   1:  PR[GP1:91,2] = PR[GP1:90,2] + -18.004;
   1:L PR[91] R[100]mm/sec CNT100;
   1:  PR[GP1:91,1] = PR[GP1:90,1] + -44.967;
   1:  PR[GP1:91,2] = PR[GP1:90,2] + -27.584;
   1:L PR[91] R[100]mm/sec CNT100;
   1:  PR[GP1:91,1] = PR[GP1:90,1] + -42.334;
   1:  PR[GP1:91,2] = PR[GP1:90,2] + -29.755;
   1:L PR[91] R[100]mm/sec CNT100;
   1:  PR[GP1:91,1] = PR[GP1:90,1] + -32.989;
   1:  PR[GP1:91,2] = PR[GP1:90,2] + -37.151;
   1:L PR[91] R[100]mm/sec CNT100;
   1:  PR[GP1:91,1] = PR[GP1:90,1] + -30.364;
   1:  PR[GP1:91,2] = PR[GP1:90,2] + -38.119;
   1:L PR[91] R[100]mm/sec CNT100;
   1:  PR[GP1:91,1] = PR[GP1:90,1] + -18.205;
   1:  PR[GP1:91,2] = PR[GP1:90,2] + -42.108;
   1:L PR[91] R[100]mm/sec CNT100;
   1:  PR[GP1:91,1] = PR[GP1:90,1] + -16.121;
   1:  PR[GP1:91,2] = PR[GP1:90,2] + -42.145;
   1:L PR[91] R[100]mm/sec CNT100;
   1:  PR[GP1:91,1] = PR[GP1:90,1] + -2.431;
   1:  PR[GP1:91,2] = PR[GP1:90,2] + -41.656;
   1:L PR[91] R[100]mm/sec CNT100;
   1:  PR[GP1:91,1] = PR[GP1:90,1] + -1.102;
   1:  PR[GP1:91,2] = PR[GP1:90,2] + -41.254;
   1:L PR[91] R[100]mm/sec CNT100;
   1:  PR[GP1:91,1] = PR[GP1:90,1] + 1.318;
   1:L PR[91] R[100]mm/sec CNT100;
   1:  PR[GP1:91,1] = PR[GP1:90,1] + 2.646;
   1:  PR[GP1:91,2] = PR[GP1:90,2] + -41.656;
   1:L PR[91] R[100]mm/sec CNT100;
   1:  PR[GP1:91,1] = PR[GP1:90,1] + 16.336;
   1:  PR[GP1:91,2] = PR[GP1:90,2] + -42.144;
   1:L PR[91] R[100]mm/sec CNT100;
   1:  PR[GP1:91,1] = PR[GP1:90,1] + 18.420;
   1:  PR[GP1:91,2] = PR[GP1:90,2] + -42.107;
   1:L PR[91] R[100]mm/sec CNT100;
   1:  PR[GP1:91,1] = PR[GP1:90,1] + 30.578;
   1:  PR[GP1:91,2] = PR[GP1:90,2] + -38.119;
   1:L PR[91] R[100]mm/sec CNT100;
   1:  PR[GP1:91,1] = PR[GP1:90,1] + 33.204;
   1:  PR[GP1:91,2] = PR[GP1:90,2] + -37.151;
   1:L PR[91] R[100]mm/sec CNT100;
   1:  PR[GP1:91,1] = PR[GP1:90,1] + 42.548;
   1:  PR[GP1:91,2] = PR[GP1:90,2] + -29.754;
   1:L PR[91] R[100]mm/sec CNT100;
   1:  PR[GP1:91,1] = PR[GP1:90,1] + 45.181;
   1:  PR[GP1:91,2] = PR[GP1:90,2] + -27.580;
   1:L PR[91] R[100]mm/sec CNT100;
   1:  PR[GP1:91,1] = PR[GP1:90,1] + 50.972;
   1:  PR[GP1:91,2] = PR[GP1:90,2] + -18.005;
   1:L PR[91] R[100]mm/sec CNT100;
   1:  PR[GP1:91,1] = PR[GP1:90,1] + 52.939;
   1:  PR[GP1:91,2] = PR[GP1:90,2] + -14.686;
   1:L PR[91] R[100]mm/sec CNT100;
   1:  PR[GP1:91,1] = PR[GP1:90,1] + 53.674;
   1:  PR[GP1:91,2] = PR[GP1:90,2] + -10.625;
   1:L PR[91] R[100]mm/sec CNT100;
   1:  PR[GP1:91,1] = PR[GP1:90,1] + 54.569;
   1:  PR[GP1:91,2] = PR[GP1:90,2] + -5.071;
   1:L PR[91] R[100]mm/sec CNT100;
   1:  PR[GP1:91,1] = PR[GP1:90,1] + 55.491;
   1:  PR[GP1:91,2] = PR[GP1:90,2] + -0.062;
   1:L PR[91] R[100]mm/sec CNT100;
   1:  PR[GP1:91,1] = PR[GP1:90,1] + 54.883;
   1:  PR[GP1:91,2] = PR[GP1:90,2] + 4.006;
   1:L PR[91] R[100]mm/sec CNT100;
   1:  PR[GP1:91,1] = PR[GP1:90,1] + 52.939;
   1:  PR[GP1:91,2] = PR[GP1:90,2] + 14.540;
   1:L PR[91] R[100]mm/sec CNT100;
   1:  PR[GP1:91,1] = PR[GP1:90,1] + 50.974;
   1:  PR[GP1:91,2] = PR[GP1:90,2] + 17.860;
   1:L PR[91] R[100]mm/sec CNT100;
   1:  PR[GP1:91,1] = PR[GP1:90,1] + 45.181;
   1:  PR[GP1:91,2] = PR[GP1:90,2] + 27.435;
   1:L PR[91] R[100]mm/sec CNT100;
   1:  PR[GP1:91,1] = PR[GP1:90,1] + 42.550;
   1:  PR[GP1:91,2] = PR[GP1:90,2] + 29.610;
   1:L PR[91] R[100]mm/sec CNT100;
   1:  PR[GP1:91,1] = PR[GP1:90,1] + 33.204;
   1:  PR[GP1:91,2] = PR[GP1:90,2] + 37.007;
   1:L PR[91] R[100]mm/sec CNT100;
   1:  PR[GP1:91,1] = PR[GP1:90,1] + 30.579;
   1:  PR[GP1:91,2] = PR[GP1:90,2] + 37.975;
   1:L PR[91] R[100]mm/sec CNT100;
   1:  PR[GP1:91,1] = PR[GP1:90,1] + 18.419;
   1:  PR[GP1:91,2] = PR[GP1:90,2] + 41.964;
   1:L PR[91] R[100]mm/sec CNT100;
   1:  PR[GP1:91,1] = PR[GP1:90,1] + 16.336;
   1:  PR[GP1:91,2] = PR[GP1:90,2] + 42.001;
   1:L PR[91] R[100]mm/sec CNT100;
   1:  PR[GP1:91,1] = PR[GP1:90,1] + 2.640;
   1:  PR[GP1:91,2] = PR[GP1:90,2] + 41.510;
   1:L PR[91] R[100]mm/sec CNT100;
   1:  PR[GP1:91,1] = PR[GP1:90,1] + 1.317;
   1:  PR[GP1:91,2] = PR[GP1:90,2] + 41.113;
   1:L PR[91] R[100]mm/sec CNT100;
   1:  ! -- Layer/Ebene 159 -- !;
   1:  PR[91] = PR[90];
   1:  PR[GP1:91,1] = PR[GP1:90,1] + -1.075;
   1:  PR[GP1:91,2] = PR[GP1:90,2] + 41.286;
   1:  PR[GP1:91,3] = PR[GP1:90,3] + 97.295;
   1:L PR[91] R[100]mm/sec CNT100;
   1:  PR[GP1:91,1] = PR[GP1:90,1] + -2.125;
   1:  PR[GP1:91,2] = PR[GP1:90,2] + 41.599;
   1:L PR[91] R[100]mm/sec CNT100;
   1:  PR[GP1:91,1] = PR[GP1:90,1] + -16.159;
   1:  PR[GP1:91,2] = PR[GP1:90,2] + 42.102;
   1:L PR[91] R[100]mm/sec CNT100;
   1:  PR[GP1:91,1] = PR[GP1:90,1] + -17.943;
   1:  PR[GP1:91,2] = PR[GP1:90,2] + 42.070;
   1:L PR[91] R[100]mm/sec CNT100;
   1:  PR[GP1:91,1] = PR[GP1:90,1] + -30.434;
   1:  PR[GP1:91,2] = PR[GP1:90,2] + 37.973;
   1:L PR[91] R[100]mm/sec CNT100;
   1:  PR[GP1:91,1] = PR[GP1:90,1] + -32.768;
   1:  PR[GP1:91,2] = PR[GP1:90,2] + 37.112;
   1:L PR[91] R[100]mm/sec CNT100;
   1:  PR[GP1:91,1] = PR[GP1:90,1] + -42.396;
   1:  PR[GP1:91,2] = PR[GP1:90,2] + 29.493;
   1:L PR[91] R[100]mm/sec CNT100;
   1:  PR[GP1:91,1] = PR[GP1:90,1] + -44.783;
   1:  PR[GP1:91,2] = PR[GP1:90,2] + 27.523;
   1:L PR[91] R[100]mm/sec CNT100;
   1:  PR[GP1:91,1] = PR[GP1:90,1] + -50.767;
   1:  PR[GP1:91,2] = PR[GP1:90,2] + 17.626;
   1:L PR[91] R[100]mm/sec CNT100;
   1:  PR[GP1:91,1] = PR[GP1:90,1] + -52.567;
   1:  PR[GP1:91,2] = PR[GP1:90,2] + 14.580;
   1:L PR[91] R[100]mm/sec CNT100;
   1:  PR[GP1:91,1] = PR[GP1:90,1] + -53.240;
   1:  PR[GP1:91,2] = PR[GP1:90,2] + 10.867;
   1:L PR[91] R[100]mm/sec CNT100;
   1:  PR[GP1:91,1] = PR[GP1:90,1] + -54.062;
   1:  PR[GP1:91,2] = PR[GP1:90,2] + 5.768;
   1:L PR[91] R[100]mm/sec CNT100;
   1:  PR[GP1:91,1] = PR[GP1:90,1] + -55.139;
   1:  PR[GP1:91,2] = PR[GP1:90,2] + -0.082;
   1:L PR[91] R[100]mm/sec CNT100;
   1:  PR[GP1:91,1] = PR[GP1:90,1] + -54.579;
   1:  PR[GP1:91,2] = PR[GP1:90,2] + -3.819;
   1:L PR[91] R[100]mm/sec CNT100;
   1:  PR[GP1:91,1] = PR[GP1:90,1] + -52.567;
   1:  PR[GP1:91,2] = PR[GP1:90,2] + -14.723;
   1:L PR[91] R[100]mm/sec CNT100;
   1:  PR[GP1:91,1] = PR[GP1:90,1] + -50.766;
   1:  PR[GP1:91,2] = PR[GP1:90,2] + -17.771;
   1:L PR[91] R[100]mm/sec CNT100;
   1:  PR[GP1:91,1] = PR[GP1:90,1] + -44.782;
   1:  PR[GP1:91,2] = PR[GP1:90,2] + -27.668;
   1:L PR[91] R[100]mm/sec CNT100;
   1:  PR[GP1:91,1] = PR[GP1:90,1] + -42.395;
   1:  PR[GP1:91,2] = PR[GP1:90,2] + -29.637;
   1:L PR[91] R[100]mm/sec CNT100;
   1:  PR[GP1:91,1] = PR[GP1:90,1] + -32.768;
   1:  PR[GP1:91,2] = PR[GP1:90,2] + -37.256;
   1:L PR[91] R[100]mm/sec CNT100;
   1:  PR[GP1:91,1] = PR[GP1:90,1] + -30.433;
   1:  PR[GP1:91,2] = PR[GP1:90,2] + -38.117;
   1:L PR[91] R[100]mm/sec CNT100;
   1:  PR[GP1:91,1] = PR[GP1:90,1] + -17.944;
   1:  PR[GP1:91,2] = PR[GP1:90,2] + -42.214;
   1:L PR[91] R[100]mm/sec CNT100;
   1:  PR[GP1:91,1] = PR[GP1:90,1] + -16.160;
   1:  PR[GP1:91,2] = PR[GP1:90,2] + -42.245;
   1:L PR[91] R[100]mm/sec CNT100;
   1:  PR[GP1:91,1] = PR[GP1:90,1] + -2.133;
   1:  PR[GP1:91,2] = PR[GP1:90,2] + -41.745;
   1:L PR[91] R[100]mm/sec CNT100;
   1:  PR[GP1:91,1] = PR[GP1:90,1] + -1.076;
   1:  PR[GP1:91,2] = PR[GP1:90,2] + -41.428;
   1:L PR[91] R[100]mm/sec CNT100;
   1:  PR[GP1:91,1] = PR[GP1:90,1] + 1.292;
   1:L PR[91] R[100]mm/sec CNT100;
   1:  PR[GP1:91,1] = PR[GP1:90,1] + 2.349;
   1:  PR[GP1:91,2] = PR[GP1:90,2] + -41.745;
   1:L PR[91] R[100]mm/sec CNT100;
   1:  PR[GP1:91,1] = PR[GP1:90,1] + 16.375;
   1:  PR[GP1:91,2] = PR[GP1:90,2] + -42.245;
   1:L PR[91] R[100]mm/sec CNT100;
   1:  PR[GP1:91,1] = PR[GP1:90,1] + 18.159;
   1:  PR[GP1:91,2] = PR[GP1:90,2] + -42.214;
   1:L PR[91] R[100]mm/sec CNT100;
   1:  PR[GP1:91,1] = PR[GP1:90,1] + 30.647;
   1:  PR[GP1:91,2] = PR[GP1:90,2] + -38.116;
   1:L PR[91] R[100]mm/sec CNT100;
   1:  PR[GP1:91,1] = PR[GP1:90,1] + 32.982;
   1:  PR[GP1:91,2] = PR[GP1:90,2] + -37.256;
   1:L PR[91] R[100]mm/sec CNT100;
   1:  PR[GP1:91,1] = PR[GP1:90,1] + 42.608;
   1:  PR[GP1:91,2] = PR[GP1:90,2] + -29.636;
   1:L PR[91] R[100]mm/sec CNT100;
   1:  PR[GP1:91,1] = PR[GP1:90,1] + 44.996;
   1:  PR[GP1:91,2] = PR[GP1:90,2] + -27.664;
   1:L PR[91] R[100]mm/sec CNT100;
   1:  PR[GP1:91,1] = PR[GP1:90,1] + 50.980;
   1:  PR[GP1:91,2] = PR[GP1:90,2] + -17.772;
   1:L PR[91] R[100]mm/sec CNT100;
   1:  PR[GP1:91,1] = PR[GP1:90,1] + 52.780;
   1:  PR[GP1:91,2] = PR[GP1:90,2] + -14.733;
   1:L PR[91] R[100]mm/sec CNT100;
   1:  PR[GP1:91,1] = PR[GP1:90,1] + 53.454;
   1:  PR[GP1:91,2] = PR[GP1:90,2] + -11.014;
   1:L PR[91] R[100]mm/sec CNT100;
   1:  PR[GP1:91,1] = PR[GP1:90,1] + 54.276;
   1:  PR[GP1:91,2] = PR[GP1:90,2] + -5.913;
   1:L PR[91] R[100]mm/sec CNT100;
   1:  PR[GP1:91,1] = PR[GP1:90,1] + 55.352;
   1:  PR[GP1:91,2] = PR[GP1:90,2] + -0.062;
   1:L PR[91] R[100]mm/sec CNT100;
   1:  PR[GP1:91,1] = PR[GP1:90,1] + 54.793;
   1:  PR[GP1:91,2] = PR[GP1:90,2] + 3.680;
   1:L PR[91] R[100]mm/sec CNT100;
   1:  PR[GP1:91,1] = PR[GP1:90,1] + 52.781;
   1:  PR[GP1:91,2] = PR[GP1:90,2] + 14.587;
   1:L PR[91] R[100]mm/sec CNT100;
   1:  PR[GP1:91,1] = PR[GP1:90,1] + 50.981;
   1:  PR[GP1:91,2] = PR[GP1:90,2] + 17.627;
   1:L PR[91] R[100]mm/sec CNT100;
   1:  PR[GP1:91,1] = PR[GP1:90,1] + 44.997;
   1:  PR[GP1:91,2] = PR[GP1:90,2] + 27.520;
   1:L PR[91] R[100]mm/sec CNT100;
   1:  PR[GP1:91,1] = PR[GP1:90,1] + 42.609;
   1:  PR[GP1:91,2] = PR[GP1:90,2] + 29.492;
   1:L PR[91] R[100]mm/sec CNT100;
   1:  PR[GP1:91,1] = PR[GP1:90,1] + 32.982;
   1:  PR[GP1:91,2] = PR[GP1:90,2] + 37.112;
   1:L PR[91] R[100]mm/sec CNT100;
   1:  PR[GP1:91,1] = PR[GP1:90,1] + 30.648;
   1:  PR[GP1:91,2] = PR[GP1:90,2] + 37.973;
   1:L PR[91] R[100]mm/sec CNT100;
   1:  PR[GP1:91,1] = PR[GP1:90,1] + 18.158;
   1:  PR[GP1:91,2] = PR[GP1:90,2] + 42.070;
   1:L PR[91] R[100]mm/sec CNT100;
   1:  PR[GP1:91,1] = PR[GP1:90,1] + 16.374;
   1:  PR[GP1:91,2] = PR[GP1:90,2] + 42.102;
   1:L PR[91] R[100]mm/sec CNT100;
   1:  PR[GP1:91,1] = PR[GP1:90,1] + 2.341;
   1:  PR[GP1:91,2] = PR[GP1:90,2] + 41.599;
   1:L PR[91] R[100]mm/sec CNT100;
   1:  PR[GP1:91,1] = PR[GP1:90,1] + 1.291;
   1:  PR[GP1:91,2] = PR[GP1:90,2] + 41.286;
   1:L PR[91] R[100]mm/sec CNT100;
   1:  ! -- Layer/Ebene 160 -- !;
   1:  PR[91] = PR[90];
   1:  PR[GP1:91,1] = PR[GP1:90,1] + -1.048;
   1:  PR[GP1:91,2] = PR[GP1:90,2] + 41.460;
   1:  PR[GP1:91,3] = PR[GP1:90,3] + 97.905;
   1:L PR[91] R[100]mm/sec CNT100;
   1:  PR[GP1:91,1] = PR[GP1:90,1] + -1.826;
   1:  PR[GP1:91,2] = PR[GP1:90,2] + 41.688;
   1:L PR[91] R[100]mm/sec CNT100;
   1:  PR[GP1:91,1] = PR[GP1:90,1] + -16.197;
   1:  PR[GP1:91,2] = PR[GP1:90,2] + 42.203;
   1:L PR[91] R[100]mm/sec CNT100;
   1:  PR[GP1:91,1] = PR[GP1:90,1] + -17.682;
   1:  PR[GP1:91,2] = PR[GP1:90,2] + 42.176;
   1:L PR[91] R[100]mm/sec CNT100;
   1:  PR[GP1:91,1] = PR[GP1:90,1] + -30.502;
   1:  PR[GP1:91,2] = PR[GP1:90,2] + 37.971;
   1:L PR[91] R[100]mm/sec CNT100;
   1:  PR[GP1:91,1] = PR[GP1:90,1] + -32.546;
   1:  PR[GP1:91,2] = PR[GP1:90,2] + 37.217;
   1:L PR[91] R[100]mm/sec CNT100;
   1:  PR[GP1:91,1] = PR[GP1:90,1] + -42.456;
   1:  PR[GP1:91,2] = PR[GP1:90,2] + 29.375;
   1:L PR[91] R[100]mm/sec CNT100;
   1:  PR[GP1:91,1] = PR[GP1:90,1] + -44.598;
   1:  PR[GP1:91,2] = PR[GP1:90,2] + 27.607;
   1:L PR[91] R[100]mm/sec CNT100;
   1:  PR[GP1:91,1] = PR[GP1:90,1] + -50.774;
   1:  PR[GP1:91,2] = PR[GP1:90,2] + 17.393;
   1:L PR[91] R[100]mm/sec CNT100;
   1:  PR[GP1:91,1] = PR[GP1:90,1] + -52.408;
   1:  PR[GP1:91,2] = PR[GP1:90,2] + 14.627;
   1:L PR[91] R[100]mm/sec CNT100;
   1:  PR[GP1:91,1] = PR[GP1:90,1] + -53.020;
   1:  PR[GP1:91,2] = PR[GP1:90,2] + 11.255;
   1:L PR[91] R[100]mm/sec CNT100;
   1:  PR[GP1:91,1] = PR[GP1:90,1] + -53.768;
   1:  PR[GP1:91,2] = PR[GP1:90,2] + 6.610;
   1:L PR[91] R[100]mm/sec CNT100;
   1:  PR[GP1:91,1] = PR[GP1:90,1] + -55.000;
   1:  PR[GP1:91,2] = PR[GP1:90,2] + -0.082;
   1:L PR[91] R[100]mm/sec CNT100;
   1:  PR[GP1:91,1] = PR[GP1:90,1] + -54.490;
   1:  PR[GP1:91,2] = PR[GP1:90,2] + -3.494;
   1:L PR[91] R[100]mm/sec CNT100;
   1:  PR[GP1:91,1] = PR[GP1:90,1] + -52.409;
   1:  PR[GP1:91,2] = PR[GP1:90,2] + -14.771;
   1:L PR[91] R[100]mm/sec CNT100;
   1:  PR[GP1:91,1] = PR[GP1:90,1] + -50.773;
   1:  PR[GP1:91,2] = PR[GP1:90,2] + -17.538;
   1:L PR[91] R[100]mm/sec CNT100;
   1:  PR[GP1:91,1] = PR[GP1:90,1] + -44.598;
   1:  PR[GP1:91,2] = PR[GP1:90,2] + -27.751;
   1:L PR[91] R[100]mm/sec CNT100;
   1:  PR[GP1:91,1] = PR[GP1:90,1] + -42.455;
   1:  PR[GP1:91,2] = PR[GP1:90,2] + -29.519;
   1:L PR[91] R[100]mm/sec CNT100;
   1:  PR[GP1:91,1] = PR[GP1:90,1] + -32.547;
   1:  PR[GP1:91,2] = PR[GP1:90,2] + -37.361;
   1:L PR[91] R[100]mm/sec CNT100;
   1:  PR[GP1:91,1] = PR[GP1:90,1] + -30.502;
   1:  PR[GP1:91,2] = PR[GP1:90,2] + -38.115;
   1:L PR[91] R[100]mm/sec CNT100;
   1:  PR[GP1:91,1] = PR[GP1:90,1] + -17.683;
   1:  PR[GP1:91,2] = PR[GP1:90,2] + -42.320;
   1:L PR[91] R[100]mm/sec CNT100;
   1:  PR[GP1:91,1] = PR[GP1:90,1] + -16.198;
   1:  PR[GP1:91,2] = PR[GP1:90,2] + -42.346;
   1:L PR[91] R[100]mm/sec CNT100;
   1:  PR[GP1:91,1] = PR[GP1:90,1] + -1.835;
   1:  PR[GP1:91,2] = PR[GP1:90,2] + -41.834;
   1:L PR[91] R[100]mm/sec CNT100;
   1:  PR[GP1:91,1] = PR[GP1:90,1] + -1.050;
   1:  PR[GP1:91,2] = PR[GP1:90,2] + -41.601;
   1:L PR[91] R[100]mm/sec CNT100;
   1:  PR[GP1:91,1] = PR[GP1:90,1] + 1.266;
   1:L PR[91] R[100]mm/sec CNT100;
   1:  PR[GP1:91,1] = PR[GP1:90,1] + 2.051;
   1:  PR[GP1:91,2] = PR[GP1:90,2] + -41.834;
   1:L PR[91] R[100]mm/sec CNT100;
   1:  PR[GP1:91,1] = PR[GP1:90,1] + 16.413;
   1:  PR[GP1:91,2] = PR[GP1:90,2] + -42.346;
   1:L PR[91] R[100]mm/sec CNT100;
   1:  PR[GP1:91,1] = PR[GP1:90,1] + 17.899;
   1:  PR[GP1:91,2] = PR[GP1:90,2] + -42.320;
   1:L PR[91] R[100]mm/sec CNT100;
   1:  PR[GP1:91,1] = PR[GP1:90,1] + 30.716;
   1:  PR[GP1:91,2] = PR[GP1:90,2] + -38.114;
   1:L PR[91] R[100]mm/sec CNT100;
   1:  PR[GP1:91,1] = PR[GP1:90,1] + 32.761;
   1:  PR[GP1:91,2] = PR[GP1:90,2] + -37.361;
   1:L PR[91] R[100]mm/sec CNT100;
   1:  PR[GP1:91,1] = PR[GP1:90,1] + 42.668;
   1:  PR[GP1:91,2] = PR[GP1:90,2] + -29.518;
   1:L PR[91] R[100]mm/sec CNT100;
   1:  PR[GP1:91,1] = PR[GP1:90,1] + 44.812;
   1:  PR[GP1:91,2] = PR[GP1:90,2] + -27.748;
   1:L PR[91] R[100]mm/sec CNT100;
   1:  PR[GP1:91,1] = PR[GP1:90,1] + 50.987;
   1:  PR[GP1:91,2] = PR[GP1:90,2] + -17.539;
   1:L PR[91] R[100]mm/sec CNT100;
   1:  PR[GP1:91,1] = PR[GP1:90,1] + 52.622;
   1:  PR[GP1:91,2] = PR[GP1:90,2] + -14.779;
   1:L PR[91] R[100]mm/sec CNT100;
   1:  PR[GP1:91,1] = PR[GP1:90,1] + 53.234;
   1:  PR[GP1:91,2] = PR[GP1:90,2] + -11.402;
   1:L PR[91] R[100]mm/sec CNT100;
   1:  PR[GP1:91,1] = PR[GP1:90,1] + 53.982;
   1:  PR[GP1:91,2] = PR[GP1:90,2] + -6.756;
   1:L PR[91] R[100]mm/sec CNT100;
   1:  PR[GP1:91,1] = PR[GP1:90,1] + 55.214;
   1:  PR[GP1:91,2] = PR[GP1:90,2] + -0.062;
   1:L PR[91] R[100]mm/sec CNT100;
   1:  PR[GP1:91,1] = PR[GP1:90,1] + 54.703;
   1:  PR[GP1:91,2] = PR[GP1:90,2] + 3.354;
   1:L PR[91] R[100]mm/sec CNT100;
   1:  PR[GP1:91,1] = PR[GP1:90,1] + 52.622;
   1:  PR[GP1:91,2] = PR[GP1:90,2] + 14.634;
   1:L PR[91] R[100]mm/sec CNT100;
   1:  PR[GP1:91,1] = PR[GP1:90,1] + 50.988;
   1:  PR[GP1:91,2] = PR[GP1:90,2] + 17.395;
   1:L PR[91] R[100]mm/sec CNT100;
   1:  PR[GP1:91,1] = PR[GP1:90,1] + 44.812;
   1:  PR[GP1:91,2] = PR[GP1:90,2] + 27.604;
   1:L PR[91] R[100]mm/sec CNT100;
   1:  PR[GP1:91,1] = PR[GP1:90,1] + 42.669;
   1:  PR[GP1:91,2] = PR[GP1:90,2] + 29.374;
   1:L PR[91] R[100]mm/sec CNT100;
   1:  PR[GP1:91,1] = PR[GP1:90,1] + 32.761;
   1:  PR[GP1:91,2] = PR[GP1:90,2] + 37.217;
   1:L PR[91] R[100]mm/sec CNT100;
   1:  PR[GP1:91,1] = PR[GP1:90,1] + 30.716;
   1:  PR[GP1:91,2] = PR[GP1:90,2] + 37.971;
   1:L PR[91] R[100]mm/sec CNT100;
   1:  PR[GP1:91,1] = PR[GP1:90,1] + 17.897;
   1:  PR[GP1:91,2] = PR[GP1:90,2] + 42.176;
   1:L PR[91] R[100]mm/sec CNT100;
   1:  PR[GP1:91,1] = PR[GP1:90,1] + 16.412;
   1:  PR[GP1:91,2] = PR[GP1:90,2] + 42.203;
   1:L PR[91] R[100]mm/sec CNT100;
   1:  PR[GP1:91,1] = PR[GP1:90,1] + 2.043;
   1:  PR[GP1:91,2] = PR[GP1:90,2] + 41.688;
   1:L PR[91] R[100]mm/sec CNT100;
   1:  PR[GP1:91,1] = PR[GP1:90,1] + 1.265;
   1:  PR[GP1:91,2] = PR[GP1:90,2] + 41.460;
   1:L PR[91] R[100]mm/sec CNT100;
   1:  ! -- Layer/Ebene 161 -- !;
   1:  PR[91] = PR[90];
   1:  PR[GP1:91,1] = PR[GP1:90,1] + -1.020;
   1:  PR[GP1:91,2] = PR[GP1:90,2] + 41.633;
   1:  PR[GP1:91,3] = PR[GP1:90,3] + 98.515;
   1:L PR[91] R[100]mm/sec CNT100;
   1:  PR[GP1:91,1] = PR[GP1:90,1] + -1.526;
   1:  PR[GP1:91,2] = PR[GP1:90,2] + 41.776;
   1:L PR[91] R[100]mm/sec CNT100;
   1:  PR[GP1:91,1] = PR[GP1:90,1] + -16.235;
   1:  PR[GP1:91,2] = PR[GP1:90,2] + 42.304;
   1:L PR[91] R[100]mm/sec CNT100;
   1:  PR[GP1:91,1] = PR[GP1:90,1] + -17.420;
   1:  PR[GP1:91,2] = PR[GP1:90,2] + 42.282;
   1:L PR[91] R[100]mm/sec CNT100;
   1:  PR[GP1:91,1] = PR[GP1:90,1] + -30.570;
   1:  PR[GP1:91,2] = PR[GP1:90,2] + 37.969;
   1:L PR[91] R[100]mm/sec CNT100;
   1:  PR[GP1:91,1] = PR[GP1:90,1] + -32.325;
   1:  PR[GP1:91,2] = PR[GP1:90,2] + 37.322;
   1:L PR[91] R[100]mm/sec CNT100;
   1:  PR[GP1:91,1] = PR[GP1:90,1] + -42.516;
   1:  PR[GP1:91,2] = PR[GP1:90,2] + 29.258;
   1:L PR[91] R[100]mm/sec CNT100;
   1:  PR[GP1:91,1] = PR[GP1:90,1] + -44.413;
   1:  PR[GP1:91,2] = PR[GP1:90,2] + 27.691;
   1:L PR[91] R[100]mm/sec CNT100;
   1:  PR[GP1:91,1] = PR[GP1:90,1] + -50.781;
   1:  PR[GP1:91,2] = PR[GP1:90,2] + 17.160;
   1:L PR[91] R[100]mm/sec CNT100;
   1:  PR[GP1:91,1] = PR[GP1:90,1] + -52.250;
   1:  PR[GP1:91,2] = PR[GP1:90,2] + 14.674;
   1:L PR[91] R[100]mm/sec CNT100;
   1:  PR[GP1:91,1] = PR[GP1:90,1] + -52.800;
   1:  PR[GP1:91,2] = PR[GP1:90,2] + 11.643;
   1:L PR[91] R[100]mm/sec CNT100;
   1:  PR[GP1:91,1] = PR[GP1:90,1] + -53.475;
   1:  PR[GP1:91,2] = PR[GP1:90,2] + 7.453;
   1:L PR[91] R[100]mm/sec CNT100;
   1:  PR[GP1:91,1] = PR[GP1:90,1] + -54.862;
   1:  PR[GP1:91,2] = PR[GP1:90,2] + -0.082;
   1:L PR[91] R[100]mm/sec CNT100;
   1:  PR[GP1:91,1] = PR[GP1:90,1] + -54.400;
   1:  PR[GP1:91,2] = PR[GP1:90,2] + -3.168;
   1:L PR[91] R[100]mm/sec CNT100;
   1:  PR[GP1:91,1] = PR[GP1:90,1] + -52.250;
   1:  PR[GP1:91,2] = PR[GP1:90,2] + -14.818;
   1:L PR[91] R[100]mm/sec CNT100;
   1:  PR[GP1:91,1] = PR[GP1:90,1] + -50.780;
   1:  PR[GP1:91,2] = PR[GP1:90,2] + -17.305;
   1:L PR[91] R[100]mm/sec CNT100;
   1:  PR[GP1:91,1] = PR[GP1:90,1] + -44.413;
   1:  PR[GP1:91,2] = PR[GP1:90,2] + -27.835;
   1:L PR[91] R[100]mm/sec CNT100;
   1:  PR[GP1:91,1] = PR[GP1:90,1] + -42.515;
   1:  PR[GP1:91,2] = PR[GP1:90,2] + -29.402;
   1:L PR[91] R[100]mm/sec CNT100;
   1:  PR[GP1:91,1] = PR[GP1:90,1] + -32.326;
   1:  PR[GP1:91,2] = PR[GP1:90,2] + -37.466;
   1:L PR[91] R[100]mm/sec CNT100;
   1:  PR[GP1:91,1] = PR[GP1:90,1] + -30.571;
   1:  PR[GP1:91,2] = PR[GP1:90,2] + -38.112;
   1:L PR[91] R[100]mm/sec CNT100;
   1:  PR[GP1:91,1] = PR[GP1:90,1] + -17.422;
   1:  PR[GP1:91,2] = PR[GP1:90,2] + -42.426;
   1:L PR[91] R[100]mm/sec CNT100;
   1:  PR[GP1:91,1] = PR[GP1:90,1] + -16.237;
   1:  PR[GP1:91,2] = PR[GP1:90,2] + -42.447;
   1:L PR[91] R[100]mm/sec CNT100;
   1:  PR[GP1:91,1] = PR[GP1:90,1] + -1.536;
   1:  PR[GP1:91,2] = PR[GP1:90,2] + -41.922;
   1:L PR[91] R[100]mm/sec CNT100;
   1:  PR[GP1:91,1] = PR[GP1:90,1] + -1.022;
   1:  PR[GP1:91,2] = PR[GP1:90,2] + -41.775;
   1:L PR[91] R[100]mm/sec CNT100;
   1:  PR[GP1:91,1] = PR[GP1:90,1] + 1.239;
   1:L PR[91] R[100]mm/sec CNT100;
   1:  PR[GP1:91,1] = PR[GP1:90,1] + 1.752;
   1:  PR[GP1:91,2] = PR[GP1:90,2] + -41.923;
   1:L PR[91] R[100]mm/sec CNT100;
   1:  PR[GP1:91,1] = PR[GP1:90,1] + 16.452;
   1:  PR[GP1:91,2] = PR[GP1:90,2] + -42.446;
   1:L PR[91] R[100]mm/sec CNT100;
   1:  PR[GP1:91,1] = PR[GP1:90,1] + 17.638;
   1:  PR[GP1:91,2] = PR[GP1:90,2] + -42.426;
   1:L PR[91] R[100]mm/sec CNT100;
   1:  PR[GP1:91,1] = PR[GP1:90,1] + 30.785;
   1:  PR[GP1:91,2] = PR[GP1:90,2] + -38.112;
   1:L PR[91] R[100]mm/sec CNT100;
   1:  PR[GP1:91,1] = PR[GP1:90,1] + 32.540;
   1:  PR[GP1:91,2] = PR[GP1:90,2] + -37.466;
   1:L PR[91] R[100]mm/sec CNT100;
   1:  PR[GP1:91,1] = PR[GP1:90,1] + 42.728;
   1:  PR[GP1:91,2] = PR[GP1:90,2] + -29.400;
   1:L PR[91] R[100]mm/sec CNT100;
   1:  PR[GP1:91,1] = PR[GP1:90,1] + 44.627;
   1:  PR[GP1:91,2] = PR[GP1:90,2] + -27.832;
   1:L PR[91] R[100]mm/sec CNT100;
   1:  PR[GP1:91,1] = PR[GP1:90,1] + 50.994;
   1:  PR[GP1:91,2] = PR[GP1:90,2] + -17.307;
   1:L PR[91] R[100]mm/sec CNT100;
   1:  PR[GP1:91,1] = PR[GP1:90,1] + 52.463;
   1:  PR[GP1:91,2] = PR[GP1:90,2] + -14.826;
   1:L PR[91] R[100]mm/sec CNT100;
   1:  PR[GP1:91,1] = PR[GP1:90,1] + 53.013;
   1:  PR[GP1:91,2] = PR[GP1:90,2] + -11.790;
   1:L PR[91] R[100]mm/sec CNT100;
   1:  PR[GP1:91,1] = PR[GP1:90,1] + 53.688;
   1:  PR[GP1:91,2] = PR[GP1:90,2] + -7.599;
   1:L PR[91] R[100]mm/sec CNT100;
   1:  PR[GP1:91,1] = PR[GP1:90,1] + 55.075;
   1:  PR[GP1:91,2] = PR[GP1:90,2] + -0.062;
   1:L PR[91] R[100]mm/sec CNT100;
   1:  PR[GP1:91,1] = PR[GP1:90,1] + 54.613;
   1:  PR[GP1:91,2] = PR[GP1:90,2] + 3.028;
   1:L PR[91] R[100]mm/sec CNT100;
   1:  PR[GP1:91,1] = PR[GP1:90,1] + 52.464;
   1:  PR[GP1:91,2] = PR[GP1:90,2] + 14.681;
   1:L PR[91] R[100]mm/sec CNT100;
   1:  PR[GP1:91,1] = PR[GP1:90,1] + 50.995;
   1:  PR[GP1:91,2] = PR[GP1:90,2] + 17.162;
   1:L PR[91] R[100]mm/sec CNT100;
   1:  PR[GP1:91,1] = PR[GP1:90,1] + 44.627;
   1:  PR[GP1:91,2] = PR[GP1:90,2] + 27.688;
   1:L PR[91] R[100]mm/sec CNT100;
   1:  PR[GP1:91,1] = PR[GP1:90,1] + 42.729;
   1:  PR[GP1:91,2] = PR[GP1:90,2] + 29.256;
   1:L PR[91] R[100]mm/sec CNT100;
   1:  PR[GP1:91,1] = PR[GP1:90,1] + 32.539;
   1:  PR[GP1:91,2] = PR[GP1:90,2] + 37.322;
   1:L PR[91] R[100]mm/sec CNT100;
   1:  PR[GP1:91,1] = PR[GP1:90,1] + 30.785;
   1:  PR[GP1:91,2] = PR[GP1:90,2] + 37.969;
   1:L PR[91] R[100]mm/sec CNT100;
   1:  PR[GP1:91,1] = PR[GP1:90,1] + 17.636;
   1:  PR[GP1:91,2] = PR[GP1:90,2] + 42.282;
   1:L PR[91] R[100]mm/sec CNT100;
   1:  PR[GP1:91,1] = PR[GP1:90,1] + 16.451;
   1:  PR[GP1:91,2] = PR[GP1:90,2] + 42.303;
   1:L PR[91] R[100]mm/sec CNT100;
   1:  PR[GP1:91,1] = PR[GP1:90,1] + 1.742;
   1:  PR[GP1:91,2] = PR[GP1:90,2] + 41.776;
   1:L PR[91] R[100]mm/sec CNT100;
   1:  PR[GP1:91,1] = PR[GP1:90,1] + 1.237;
   1:  PR[GP1:91,2] = PR[GP1:90,2] + 41.633;
   1:L PR[91] R[100]mm/sec CNT100;
   1:  ! -- Layer/Ebene 162 -- !;
   1:  PR[91] = PR[90];
   1:  PR[GP1:91,1] = PR[GP1:90,1] + -0.992;
   1:  PR[GP1:91,2] = PR[GP1:90,2] + 41.801;
   1:  PR[GP1:91,3] = PR[GP1:90,3] + 99.125;
   1:L PR[91] R[100]mm/sec CNT100;
   1:  PR[GP1:91,1] = PR[GP1:90,1] + -1.225;
   1:  PR[GP1:91,2] = PR[GP1:90,2] + 41.865;
   1:L PR[91] R[100]mm/sec CNT100;
   1:  PR[GP1:91,1] = PR[GP1:90,1] + -16.273;
   1:  PR[GP1:91,2] = PR[GP1:90,2] + 42.404;
   1:L PR[91] R[100]mm/sec CNT100;
   1:  PR[GP1:91,1] = PR[GP1:90,1] + -17.159;
   1:  PR[GP1:91,2] = PR[GP1:90,2] + 42.388;
   1:L PR[91] R[100]mm/sec CNT100;
   1:  PR[GP1:91,1] = PR[GP1:90,1] + -30.639;
   1:  PR[GP1:91,2] = PR[GP1:90,2] + 37.967;
   1:L PR[91] R[100]mm/sec CNT100;
   1:  PR[GP1:91,1] = PR[GP1:90,1] + -32.103;
   1:  PR[GP1:91,2] = PR[GP1:90,2] + 37.427;
   1:L PR[91] R[100]mm/sec CNT100;
   1:  PR[GP1:91,1] = PR[GP1:90,1] + -42.576;
   1:  PR[GP1:91,2] = PR[GP1:90,2] + 29.140;
   1:L PR[91] R[100]mm/sec CNT100;
   1:  PR[GP1:91,1] = PR[GP1:90,1] + -44.229;
   1:  PR[GP1:91,2] = PR[GP1:90,2] + 27.776;
   1:L PR[91] R[100]mm/sec CNT100;
   1:  PR[GP1:91,1] = PR[GP1:90,1] + -50.788;
   1:  PR[GP1:91,2] = PR[GP1:90,2] + 16.928;
   1:L PR[91] R[100]mm/sec CNT100;
   1:  PR[GP1:91,1] = PR[GP1:90,1] + -52.092;
   1:  PR[GP1:91,2] = PR[GP1:90,2] + 14.722;
   1:L PR[91] R[100]mm/sec CNT100;
   1:  PR[GP1:91,1] = PR[GP1:90,1] + -52.579;
   1:  PR[GP1:91,2] = PR[GP1:90,2] + 12.031;
   1:L PR[91] R[100]mm/sec CNT100;
   1:  PR[GP1:91,1] = PR[GP1:90,1] + -53.181;
   1:  PR[GP1:91,2] = PR[GP1:90,2] + 8.295;
   1:L PR[91] R[100]mm/sec CNT100;
   1:  PR[GP1:91,1] = PR[GP1:90,1] + -54.724;
   1:  PR[GP1:91,2] = PR[GP1:90,2] + -0.082;
   1:L PR[91] R[100]mm/sec CNT100;
   1:  PR[GP1:91,1] = PR[GP1:90,1] + -54.310;
   1:  PR[GP1:91,2] = PR[GP1:90,2] + -2.842;
   1:L PR[91] R[100]mm/sec CNT100;
   1:  PR[GP1:91,1] = PR[GP1:90,1] + -52.092;
   1:  PR[GP1:91,2] = PR[GP1:90,2] + -14.865;
   1:L PR[91] R[100]mm/sec CNT100;
   1:  PR[GP1:91,1] = PR[GP1:90,1] + -50.787;
   1:  PR[GP1:91,2] = PR[GP1:90,2] + -17.072;
   1:L PR[91] R[100]mm/sec CNT100;
   1:  PR[GP1:91,1] = PR[GP1:90,1] + -44.229;
   1:  PR[GP1:91,2] = PR[GP1:90,2] + -27.919;
   1:L PR[91] R[100]mm/sec CNT100;
   1:  PR[GP1:91,1] = PR[GP1:90,1] + -42.575;
   1:  PR[GP1:91,2] = PR[GP1:90,2] + -29.284;
   1:L PR[91] R[100]mm/sec CNT100;
   1:  PR[GP1:91,1] = PR[GP1:90,1] + -32.104;
   1:  PR[GP1:91,2] = PR[GP1:90,2] + -37.570;
   1:L PR[91] R[100]mm/sec CNT100;
   1:  PR[GP1:91,1] = PR[GP1:90,1] + -30.639;
   1:  PR[GP1:91,2] = PR[GP1:90,2] + -38.110;
   1:L PR[91] R[100]mm/sec CNT100;
   1:  PR[GP1:91,1] = PR[GP1:90,1] + -17.161;
   1:  PR[GP1:91,2] = PR[GP1:90,2] + -42.532;
   1:L PR[91] R[100]mm/sec CNT100;
   1:  PR[GP1:91,1] = PR[GP1:90,1] + -16.276;
   1:  PR[GP1:91,2] = PR[GP1:90,2] + -42.547;
   1:L PR[91] R[100]mm/sec CNT100;
   1:  PR[GP1:91,1] = PR[GP1:90,1] + -1.234;
   1:  PR[GP1:91,2] = PR[GP1:90,2] + -42.011;
   1:L PR[91] R[100]mm/sec CNT100;
   1:  PR[GP1:91,1] = PR[GP1:90,1] + -0.993;
   1:  PR[GP1:91,2] = PR[GP1:90,2] + -41.946;
   1:L PR[91] R[100]mm/sec CNT100;
   1:  PR[GP1:91,1] = PR[GP1:90,1] + 1.209;
   1:L PR[91] R[100]mm/sec CNT100;
   1:  PR[GP1:91,1] = PR[GP1:90,1] + 1.451;
   1:  PR[GP1:91,2] = PR[GP1:90,2] + -42.011;
   1:L PR[91] R[100]mm/sec CNT100;
   1:  PR[GP1:91,1] = PR[GP1:90,1] + 16.491;
   1:  PR[GP1:91,2] = PR[GP1:90,2] + -42.547;
   1:L PR[91] R[100]mm/sec CNT100;
   1:  PR[GP1:91,1] = PR[GP1:90,1] + 17.377;
   1:  PR[GP1:91,2] = PR[GP1:90,2] + -42.532;
   1:L PR[91] R[100]mm/sec CNT100;
   1:  PR[GP1:91,1] = PR[GP1:90,1] + 30.854;
   1:  PR[GP1:91,2] = PR[GP1:90,2] + -38.110;
   1:L PR[91] R[100]mm/sec CNT100;
   1:  PR[GP1:91,1] = PR[GP1:90,1] + 32.319;
   1:  PR[GP1:91,2] = PR[GP1:90,2] + -37.570;
   1:L PR[91] R[100]mm/sec CNT100;
   1:  PR[GP1:91,1] = PR[GP1:90,1] + 42.789;
   1:  PR[GP1:91,2] = PR[GP1:90,2] + -29.282;
   1:L PR[91] R[100]mm/sec CNT100;
   1:  PR[GP1:91,1] = PR[GP1:90,1] + 44.443;
   1:  PR[GP1:91,2] = PR[GP1:90,2] + -27.916;
   1:L PR[91] R[100]mm/sec CNT100;
   1:  PR[GP1:91,1] = PR[GP1:90,1] + 51.001;
   1:  PR[GP1:91,2] = PR[GP1:90,2] + -17.074;
   1:L PR[91] R[100]mm/sec CNT100;
   1:  PR[GP1:91,1] = PR[GP1:90,1] + 52.305;
   1:  PR[GP1:91,2] = PR[GP1:90,2] + -14.873;
   1:L PR[91] R[100]mm/sec CNT100;
   1:  PR[GP1:91,1] = PR[GP1:90,1] + 52.793;
   1:  PR[GP1:91,2] = PR[GP1:90,2] + -12.178;
   1:L PR[91] R[100]mm/sec CNT100;
   1:  PR[GP1:91,1] = PR[GP1:90,1] + 53.395;
   1:  PR[GP1:91,2] = PR[GP1:90,2] + -8.441;
   1:L PR[91] R[100]mm/sec CNT100;
   1:  PR[GP1:91,1] = PR[GP1:90,1] + 54.937;
   1:  PR[GP1:91,2] = PR[GP1:90,2] + -0.062;
   1:L PR[91] R[100]mm/sec CNT100;
   1:  PR[GP1:91,1] = PR[GP1:90,1] + 54.524;
   1:  PR[GP1:91,2] = PR[GP1:90,2] + 2.702;
   1:L PR[91] R[100]mm/sec CNT100;
   1:  PR[GP1:91,1] = PR[GP1:90,1] + 52.305;
   1:  PR[GP1:91,2] = PR[GP1:90,2] + 14.728;
   1:L PR[91] R[100]mm/sec CNT100;
   1:  PR[GP1:91,1] = PR[GP1:90,1] + 51.002;
   1:  PR[GP1:91,2] = PR[GP1:90,2] + 16.930;
   1:L PR[91] R[100]mm/sec CNT100;
   1:  PR[GP1:91,1] = PR[GP1:90,1] + 44.443;
   1:  PR[GP1:91,2] = PR[GP1:90,2] + 27.772;
   1:L PR[91] R[100]mm/sec CNT100;
   1:  PR[GP1:91,1] = PR[GP1:90,1] + 42.789;
   1:  PR[GP1:91,2] = PR[GP1:90,2] + 29.138;
   1:L PR[91] R[100]mm/sec CNT100;
   1:  PR[GP1:91,1] = PR[GP1:90,1] + 32.318;
   1:  PR[GP1:91,2] = PR[GP1:90,2] + 37.427;
   1:L PR[91] R[100]mm/sec CNT100;
   1:  PR[GP1:91,1] = PR[GP1:90,1] + 30.853;
   1:  PR[GP1:91,2] = PR[GP1:90,2] + 37.967;
   1:L PR[91] R[100]mm/sec CNT100;
   1:  PR[GP1:91,1] = PR[GP1:90,1] + 17.375;
   1:  PR[GP1:91,2] = PR[GP1:90,2] + 42.388;
   1:L PR[91] R[100]mm/sec CNT100;
   1:  PR[GP1:91,1] = PR[GP1:90,1] + 16.489;
   1:  PR[GP1:91,2] = PR[GP1:90,2] + 42.404;
   1:L PR[91] R[100]mm/sec CNT100;
   1:  PR[GP1:91,1] = PR[GP1:90,1] + 1.442;
   1:  PR[GP1:91,2] = PR[GP1:90,2] + 41.865;
   1:L PR[91] R[100]mm/sec CNT100;
   1:  PR[GP1:91,1] = PR[GP1:90,1] + 1.209;
   1:  PR[GP1:91,2] = PR[GP1:90,2] + 41.802;
   1:L PR[91] R[100]mm/sec CNT100;
   1:  ! -- Layer/Ebene 163 -- !;
   1:  PR[91] = PR[90];
   1:  PR[GP1:91,1] = PR[GP1:90,1] + -0.897;
   1:  PR[GP1:91,2] = PR[GP1:90,2] + 41.964;
   1:  PR[GP1:91,3] = PR[GP1:90,3] + 99.735;
   1:L PR[91] R[100]mm/sec CNT100;
   1:  PR[GP1:91,1] = PR[GP1:90,1] + -2.090;
   1:  PR[GP1:91,2] = PR[GP1:90,2] + 41.995;
   1:L PR[91] R[100]mm/sec CNT100;
   1:  PR[GP1:91,1] = PR[GP1:90,1] + -16.311;
   1:  PR[GP1:91,2] = PR[GP1:90,2] + 42.505;
   1:L PR[91] R[100]mm/sec CNT100;
   1:  PR[GP1:91,1] = PR[GP1:90,1] + -16.897;
   1:  PR[GP1:91,2] = PR[GP1:90,2] + 42.494;
   1:L PR[91] R[100]mm/sec CNT100;
   1:  PR[GP1:91,1] = PR[GP1:90,1] + -30.707;
   1:  PR[GP1:91,2] = PR[GP1:90,2] + 37.965;
   1:L PR[91] R[100]mm/sec CNT100;
   1:  PR[GP1:91,1] = PR[GP1:90,1] + -31.882;
   1:  PR[GP1:91,2] = PR[GP1:90,2] + 37.532;
   1:L PR[91] R[100]mm/sec CNT100;
   1:  PR[GP1:91,1] = PR[GP1:90,1] + -42.636;
   1:  PR[GP1:91,2] = PR[GP1:90,2] + 29.022;
   1:L PR[91] R[100]mm/sec CNT100;
   1:  PR[GP1:91,1] = PR[GP1:90,1] + -44.044;
   1:  PR[GP1:91,2] = PR[GP1:90,2] + 27.860;
   1:L PR[91] R[100]mm/sec CNT100;
   1:  PR[GP1:91,1] = PR[GP1:90,1] + -50.795;
   1:  PR[GP1:91,2] = PR[GP1:90,2] + 16.694;
   1:L PR[91] R[100]mm/sec CNT100;
   1:  PR[GP1:91,1] = PR[GP1:90,1] + -51.933;
   1:  PR[GP1:91,2] = PR[GP1:90,2] + 14.769;
   1:L PR[91] R[100]mm/sec CNT100;
   1:  PR[GP1:91,1] = PR[GP1:90,1] + -52.359;
   1:  PR[GP1:91,2] = PR[GP1:90,2] + 12.419;
   1:L PR[91] R[100]mm/sec CNT100;
   1:  PR[GP1:91,1] = PR[GP1:90,1] + -52.888;
   1:  PR[GP1:91,2] = PR[GP1:90,2] + 9.138;
   1:L PR[91] R[100]mm/sec CNT100;
   1:  PR[GP1:91,1] = PR[GP1:90,1] + -54.585;
   1:  PR[GP1:91,2] = PR[GP1:90,2] + -0.082;
   1:L PR[91] R[100]mm/sec CNT100;
   1:  PR[GP1:91,1] = PR[GP1:90,1] + -54.220;
   1:  PR[GP1:91,2] = PR[GP1:90,2] + -2.517;
   1:L PR[91] R[100]mm/sec CNT100;
   1:  PR[GP1:91,1] = PR[GP1:90,1] + -51.934;
   1:  PR[GP1:91,2] = PR[GP1:90,2] + -14.912;
   1:L PR[91] R[100]mm/sec CNT100;
   1:  PR[GP1:91,1] = PR[GP1:90,1] + -50.794;
   1:  PR[GP1:91,2] = PR[GP1:90,2] + -16.839;
   1:L PR[91] R[100]mm/sec CNT100;
   1:  PR[GP1:91,1] = PR[GP1:90,1] + -44.044;
   1:  PR[GP1:91,2] = PR[GP1:90,2] + -28.003;
   1:L PR[91] R[100]mm/sec CNT100;
   1:  PR[GP1:91,1] = PR[GP1:90,1] + -42.635;
   1:  PR[GP1:91,2] = PR[GP1:90,2] + -29.166;
   1:L PR[91] R[100]mm/sec CNT100;
   1:  PR[GP1:91,1] = PR[GP1:90,1] + -31.883;
   1:  PR[GP1:91,2] = PR[GP1:90,2] + -37.675;
   1:L PR[91] R[100]mm/sec CNT100;
   1:  PR[GP1:91,1] = PR[GP1:90,1] + -30.708;
   1:  PR[GP1:91,2] = PR[GP1:90,2] + -38.108;
   1:L PR[91] R[100]mm/sec CNT100;
   1:  PR[GP1:91,1] = PR[GP1:90,1] + -16.901;
   1:  PR[GP1:91,2] = PR[GP1:90,2] + -42.638;
   1:L PR[91] R[100]mm/sec CNT100;
   1:  PR[GP1:91,1] = PR[GP1:90,1] + -16.314;
   1:  PR[GP1:91,2] = PR[GP1:90,2] + -42.648;
   1:L PR[91] R[100]mm/sec CNT100;
   1:  PR[GP1:91,1] = PR[GP1:90,1] + -0.892;
   1:  PR[GP1:91,2] = PR[GP1:90,2] + -42.108;
   1:L PR[91] R[100]mm/sec CNT100;
   1:  PR[GP1:91,1] = PR[GP1:90,1] + 1.113;
   1:L PR[91] R[100]mm/sec CNT100;
   1:  PR[GP1:91,1] = PR[GP1:90,1] + 2.088;
   1:  PR[GP1:91,2] = PR[GP1:90,2] + -42.133;
   1:L PR[91] R[100]mm/sec CNT100;
   1:  PR[GP1:91,1] = PR[GP1:90,1] + 16.530;
   1:  PR[GP1:91,2] = PR[GP1:90,2] + -42.648;
   1:L PR[91] R[100]mm/sec CNT100;
   1:  PR[GP1:91,1] = PR[GP1:90,1] + 17.116;
   1:  PR[GP1:91,2] = PR[GP1:90,2] + -42.638;
   1:L PR[91] R[100]mm/sec CNT100;
   1:  PR[GP1:91,1] = PR[GP1:90,1] + 30.923;
   1:  PR[GP1:91,2] = PR[GP1:90,2] + -38.108;
   1:L PR[91] R[100]mm/sec CNT100;
   1:  PR[GP1:91,1] = PR[GP1:90,1] + 32.098;
   1:  PR[GP1:91,2] = PR[GP1:90,2] + -37.675;
   1:L PR[91] R[100]mm/sec CNT100;
   1:  PR[GP1:91,1] = PR[GP1:90,1] + 42.849;
   1:  PR[GP1:91,2] = PR[GP1:90,2] + -29.164;
   1:L PR[91] R[100]mm/sec CNT100;
   1:  PR[GP1:91,1] = PR[GP1:90,1] + 44.258;
   1:  PR[GP1:91,2] = PR[GP1:90,2] + -28.000;
   1:L PR[91] R[100]mm/sec CNT100;
   1:  PR[GP1:91,1] = PR[GP1:90,1] + 51.008;
   1:  PR[GP1:91,2] = PR[GP1:90,2] + -16.841;
   1:L PR[91] R[100]mm/sec CNT100;
   1:  PR[GP1:91,1] = PR[GP1:90,1] + 52.146;
   1:  PR[GP1:91,2] = PR[GP1:90,2] + -14.920;
   1:L PR[91] R[100]mm/sec CNT100;
   1:  PR[GP1:91,1] = PR[GP1:90,1] + 52.573;
   1:  PR[GP1:91,2] = PR[GP1:90,2] + -12.566;
   1:L PR[91] R[100]mm/sec CNT100;
   1:  PR[GP1:91,1] = PR[GP1:90,1] + 53.101;
   1:  PR[GP1:91,2] = PR[GP1:90,2] + -9.284;
   1:L PR[91] R[100]mm/sec CNT100;
   1:  PR[GP1:91,1] = PR[GP1:90,1] + 54.798;
   1:  PR[GP1:91,2] = PR[GP1:90,2] + -0.062;
   1:L PR[91] R[100]mm/sec CNT100;
   1:  PR[GP1:91,1] = PR[GP1:90,1] + 54.434;
   1:  PR[GP1:91,2] = PR[GP1:90,2] + 2.376;
   1:L PR[91] R[100]mm/sec CNT100;
   1:  PR[GP1:91,1] = PR[GP1:90,1] + 52.147;
   1:  PR[GP1:91,2] = PR[GP1:90,2] + 14.775;
   1:L PR[91] R[100]mm/sec CNT100;
   1:  PR[GP1:91,1] = PR[GP1:90,1] + 51.009;
   1:  PR[GP1:91,2] = PR[GP1:90,2] + 16.697;
   1:L PR[91] R[100]mm/sec CNT100;
   1:  PR[GP1:91,1] = PR[GP1:90,1] + 44.258;
   1:  PR[GP1:91,2] = PR[GP1:90,2] + 27.856;
   1:L PR[91] R[100]mm/sec CNT100;
   1:  PR[GP1:91,1] = PR[GP1:90,1] + 42.849;
   1:  PR[GP1:91,2] = PR[GP1:90,2] + 29.020;
   1:L PR[91] R[100]mm/sec CNT100;
   1:  PR[GP1:91,1] = PR[GP1:90,1] + 32.097;
   1:  PR[GP1:91,2] = PR[GP1:90,2] + 37.532;
   1:L PR[91] R[100]mm/sec CNT100;
   1:  PR[GP1:91,1] = PR[GP1:90,1] + 30.922;
   1:  PR[GP1:91,2] = PR[GP1:90,2] + 37.965;
   1:L PR[91] R[100]mm/sec CNT100;
   1:  PR[GP1:91,1] = PR[GP1:90,1] + 17.113;
   1:  PR[GP1:91,2] = PR[GP1:90,2] + 42.494;
   1:L PR[91] R[100]mm/sec CNT100;
   1:  PR[GP1:91,1] = PR[GP1:90,1] + 16.527;
   1:  PR[GP1:91,2] = PR[GP1:90,2] + 42.505;
   1:L PR[91] R[100]mm/sec CNT100;
   1:  PR[GP1:91,1] = PR[GP1:90,1] + 2.301;
   1:  PR[GP1:91,2] = PR[GP1:90,2] + 41.995;
   1:L PR[91] R[100]mm/sec CNT100;
   1:  PR[GP1:91,1] = PR[GP1:90,1] + 1.104;
   1:  PR[GP1:91,2] = PR[GP1:90,2] + 41.964;
   1:L PR[91] R[100]mm/sec CNT100;
   1:  ! -- Layer/Ebene 164 -- !;
   1:  PR[91] = PR[90];
   1:  PR[GP1:91,1] = PR[GP1:90,1] + -0.875;
   1:  PR[GP1:91,2] = PR[GP1:90,2] + 42.123;
   1:  PR[GP1:91,3] = PR[GP1:90,3] + 100.345;
   1:L PR[91] R[100]mm/sec CNT100;
   1:  PR[GP1:91,1] = PR[GP1:90,1] + -8.287;
   1:  PR[GP1:91,2] = PR[GP1:90,2] + 42.316;
   1:L PR[91] R[100]mm/sec CNT100;
   1:  PR[GP1:91,1] = PR[GP1:90,1] + -16.350;
   1:  PR[GP1:91,2] = PR[GP1:90,2] + 42.606;
   1:L PR[91] R[100]mm/sec CNT100;
   1:  PR[GP1:91,1] = PR[GP1:90,1] + -16.636;
   1:  PR[GP1:91,2] = PR[GP1:90,2] + 42.600;
   1:L PR[91] R[100]mm/sec CNT100;
   1:  PR[GP1:91,1] = PR[GP1:90,1] + -30.776;
   1:  PR[GP1:91,2] = PR[GP1:90,2] + 37.963;
   1:L PR[91] R[100]mm/sec CNT100;
   1:  PR[GP1:91,1] = PR[GP1:90,1] + -31.660;
   1:  PR[GP1:91,2] = PR[GP1:90,2] + 37.637;
   1:L PR[91] R[100]mm/sec CNT100;
   1:  PR[GP1:91,1] = PR[GP1:90,1] + -42.695;
   1:  PR[GP1:91,2] = PR[GP1:90,2] + 28.905;
   1:L PR[91] R[100]mm/sec CNT100;
   1:  PR[GP1:91,1] = PR[GP1:90,1] + -43.859;
   1:  PR[GP1:91,2] = PR[GP1:90,2] + 27.944;
   1:L PR[91] R[100]mm/sec CNT100;
   1:  PR[GP1:91,1] = PR[GP1:90,1] + -50.802;
   1:  PR[GP1:91,2] = PR[GP1:90,2] + 16.462;
   1:L PR[91] R[100]mm/sec CNT100;
   1:  PR[GP1:91,1] = PR[GP1:90,1] + -51.774;
   1:  PR[GP1:91,2] = PR[GP1:90,2] + 14.816;
   1:L PR[91] R[100]mm/sec CNT100;
   1:  PR[GP1:91,1] = PR[GP1:90,1] + -52.139;
   1:  PR[GP1:91,2] = PR[GP1:90,2] + 12.807;
   1:L PR[91] R[100]mm/sec CNT100;
   1:  PR[GP1:91,1] = PR[GP1:90,1] + -52.594;
   1:  PR[GP1:91,2] = PR[GP1:90,2] + 9.981;
   1:L PR[91] R[100]mm/sec CNT100;
   1:  PR[GP1:91,1] = PR[GP1:90,1] + -54.447;
   1:  PR[GP1:91,2] = PR[GP1:90,2] + -0.082;
   1:L PR[91] R[100]mm/sec CNT100;
   1:  PR[GP1:91,1] = PR[GP1:90,1] + -54.131;
   1:  PR[GP1:91,2] = PR[GP1:90,2] + -2.191;
   1:L PR[91] R[100]mm/sec CNT100;
   1:  PR[GP1:91,1] = PR[GP1:90,1] + -51.775;
   1:  PR[GP1:91,2] = PR[GP1:90,2] + -14.959;
   1:L PR[91] R[100]mm/sec CNT100;
   1:  PR[GP1:91,1] = PR[GP1:90,1] + -50.801;
   1:  PR[GP1:91,2] = PR[GP1:90,2] + -16.606;
   1:L PR[91] R[100]mm/sec CNT100;
   1:  PR[GP1:91,1] = PR[GP1:90,1] + -43.860;
   1:  PR[GP1:91,2] = PR[GP1:90,2] + -28.087;
   1:L PR[91] R[100]mm/sec CNT100;
   1:  PR[GP1:91,1] = PR[GP1:90,1] + -42.695;
   1:  PR[GP1:91,2] = PR[GP1:90,2] + -29.048;
   1:L PR[91] R[100]mm/sec CNT100;
   1:  PR[GP1:91,1] = PR[GP1:90,1] + -31.662;
   1:  PR[GP1:91,2] = PR[GP1:90,2] + -37.780;
   1:L PR[91] R[100]mm/sec CNT100;
   1:  PR[GP1:91,1] = PR[GP1:90,1] + -30.777;
   1:  PR[GP1:91,2] = PR[GP1:90,2] + -38.106;
   1:L PR[91] R[100]mm/sec CNT100;
   1:  PR[GP1:91,1] = PR[GP1:90,1] + -16.640;
   1:  PR[GP1:91,2] = PR[GP1:90,2] + -42.744;
   1:L PR[91] R[100]mm/sec CNT100;
   1:  PR[GP1:91,1] = PR[GP1:90,1] + -16.353;
   1:  PR[GP1:91,2] = PR[GP1:90,2] + -42.749;
   1:L PR[91] R[100]mm/sec CNT100;
   1:  PR[GP1:91,1] = PR[GP1:90,1] + -8.166;
   1:  PR[GP1:91,2] = PR[GP1:90,2] + -42.457;
   1:L PR[91] R[100]mm/sec CNT100;
   1:  PR[GP1:91,1] = PR[GP1:90,1] + -0.874;
   1:  PR[GP1:91,2] = PR[GP1:90,2] + -42.267;
   1:L PR[91] R[100]mm/sec CNT100;
   1:  PR[GP1:91,1] = PR[GP1:90,1] + 1.090;
   1:L PR[91] R[100]mm/sec CNT100;
   1:  PR[GP1:91,1] = PR[GP1:90,1] + 8.377;
   1:  PR[GP1:91,2] = PR[GP1:90,2] + -42.457;
   1:L PR[91] R[100]mm/sec CNT100;
   1:  PR[GP1:91,1] = PR[GP1:90,1] + 16.569;
   1:  PR[GP1:91,2] = PR[GP1:90,2] + -42.749;
   1:L PR[91] R[100]mm/sec CNT100;
   1:  PR[GP1:91,1] = PR[GP1:90,1] + 16.856;
   1:  PR[GP1:91,2] = PR[GP1:90,2] + -42.744;
   1:L PR[91] R[100]mm/sec CNT100;
   1:  PR[GP1:91,1] = PR[GP1:90,1] + 30.992;
   1:  PR[GP1:91,2] = PR[GP1:90,2] + -38.106;
   1:L PR[91] R[100]mm/sec CNT100;
   1:  PR[GP1:91,1] = PR[GP1:90,1] + 31.877;
   1:  PR[GP1:91,2] = PR[GP1:90,2] + -37.780;
   1:L PR[91] R[100]mm/sec CNT100;
   1:  PR[GP1:91,1] = PR[GP1:90,1] + 42.909;
   1:  PR[GP1:91,2] = PR[GP1:90,2] + -29.046;
   1:L PR[91] R[100]mm/sec CNT100;
   1:  PR[GP1:91,1] = PR[GP1:90,1] + 44.074;
   1:  PR[GP1:91,2] = PR[GP1:90,2] + -28.084;
   1:L PR[91] R[100]mm/sec CNT100;
   1:  PR[GP1:91,1] = PR[GP1:90,1] + 51.015;
   1:  PR[GP1:91,2] = PR[GP1:90,2] + -16.609;
   1:L PR[91] R[100]mm/sec CNT100;
   1:  PR[GP1:91,1] = PR[GP1:90,1] + 51.988;
   1:  PR[GP1:91,2] = PR[GP1:90,2] + -14.966;
   1:L PR[91] R[100]mm/sec CNT100;
   1:  PR[GP1:91,1] = PR[GP1:90,1] + 52.352;
   1:  PR[GP1:91,2] = PR[GP1:90,2] + -12.955;
   1:L PR[91] R[100]mm/sec CNT100;
   1:  PR[GP1:91,1] = PR[GP1:90,1] + 52.808;
   1:  PR[GP1:91,2] = PR[GP1:90,2] + -10.127;
   1:L PR[91] R[100]mm/sec CNT100;
   1:  PR[GP1:91,1] = PR[GP1:90,1] + 54.660;
   1:  PR[GP1:91,2] = PR[GP1:90,2] + -0.062;
   1:L PR[91] R[100]mm/sec CNT100;
   1:  PR[GP1:91,1] = PR[GP1:90,1] + 54.344;
   1:  PR[GP1:91,2] = PR[GP1:90,2] + 2.050;
   1:L PR[91] R[100]mm/sec CNT100;
   1:  PR[GP1:91,1] = PR[GP1:90,1] + 51.988;
   1:  PR[GP1:91,2] = PR[GP1:90,2] + 14.822;
   1:L PR[91] R[100]mm/sec CNT100;
   1:  PR[GP1:91,1] = PR[GP1:90,1] + 51.016;
   1:  PR[GP1:91,2] = PR[GP1:90,2] + 16.465;
   1:L PR[91] R[100]mm/sec CNT100;
   1:  PR[GP1:91,1] = PR[GP1:90,1] + 44.073;
   1:  PR[GP1:91,2] = PR[GP1:90,2] + 27.941;
   1:L PR[91] R[100]mm/sec CNT100;
   1:  PR[GP1:91,1] = PR[GP1:90,1] + 42.909;
   1:  PR[GP1:91,2] = PR[GP1:90,2] + 28.903;
   1:L PR[91] R[100]mm/sec CNT100;
   1:  PR[GP1:91,1] = PR[GP1:90,1] + 31.875;
   1:  PR[GP1:91,2] = PR[GP1:90,2] + 37.637;
   1:L PR[91] R[100]mm/sec CNT100;
   1:  PR[GP1:91,1] = PR[GP1:90,1] + 30.990;
   1:  PR[GP1:91,2] = PR[GP1:90,2] + 37.963;
   1:L PR[91] R[100]mm/sec CNT100;
   1:  PR[GP1:91,1] = PR[GP1:90,1] + 16.852;
   1:  PR[GP1:91,2] = PR[GP1:90,2] + 42.600;
   1:L PR[91] R[100]mm/sec CNT100;
   1:  PR[GP1:91,1] = PR[GP1:90,1] + 16.566;
   1:  PR[GP1:91,2] = PR[GP1:90,2] + 42.605;
   1:L PR[91] R[100]mm/sec CNT100;
   1:  PR[GP1:91,1] = PR[GP1:90,1] + 8.498;
   1:  PR[GP1:91,2] = PR[GP1:90,2] + 42.316;
   1:L PR[91] R[100]mm/sec CNT100;
   1:  PR[GP1:91,1] = PR[GP1:90,1] + 1.091;
   1:  PR[GP1:91,2] = PR[GP1:90,2] + 42.123;
   1:L PR[91] R[100]mm/sec CNT100;
   1:  ! -- Layer/Ebene 165 -- !;
   1:  PR[91] = PR[90];
   1:  PR[GP1:91,1] = PR[GP1:90,1] + -0.852;
   1:  PR[GP1:91,2] = PR[GP1:90,2] + 42.282;
   1:  PR[GP1:91,3] = PR[GP1:90,3] + 100.955;
   1:L PR[91] R[100]mm/sec CNT100;
   1:  PR[GP1:91,1] = PR[GP1:90,1] + -14.482;
   1:  PR[GP1:91,2] = PR[GP1:90,2] + 42.638;
   1:L PR[91] R[100]mm/sec CNT100;
   1:  PR[GP1:91,1] = PR[GP1:90,1] + -16.390;
   1:  PR[GP1:91,2] = PR[GP1:90,2] + 42.702;
   1:L PR[91] R[100]mm/sec CNT100;
   1:  PR[GP1:91,1] = PR[GP1:90,1] + -30.844;
   1:  PR[GP1:91,2] = PR[GP1:90,2] + 37.961;
   1:L PR[91] R[100]mm/sec CNT100;
   1:  PR[GP1:91,1] = PR[GP1:90,1] + -31.439;
   1:  PR[GP1:91,2] = PR[GP1:90,2] + 37.742;
   1:L PR[91] R[100]mm/sec CNT100;
   1:  PR[GP1:91,1] = PR[GP1:90,1] + -42.755;
   1:  PR[GP1:91,2] = PR[GP1:90,2] + 28.787;
   1:L PR[91] R[100]mm/sec CNT100;
   1:  PR[GP1:91,1] = PR[GP1:90,1] + -43.675;
   1:  PR[GP1:91,2] = PR[GP1:90,2] + 28.028;
   1:L PR[91] R[100]mm/sec CNT100;
   1:  PR[GP1:91,1] = PR[GP1:90,1] + -50.809;
   1:  PR[GP1:91,2] = PR[GP1:90,2] + 16.229;
   1:L PR[91] R[100]mm/sec CNT100;
   1:  PR[GP1:91,1] = PR[GP1:90,1] + -51.616;
   1:  PR[GP1:91,2] = PR[GP1:90,2] + 14.863;
   1:L PR[91] R[100]mm/sec CNT100;
   1:  PR[GP1:91,1] = PR[GP1:90,1] + -51.918;
   1:  PR[GP1:91,2] = PR[GP1:90,2] + 13.195;
   1:L PR[91] R[100]mm/sec CNT100;
   1:  PR[GP1:91,1] = PR[GP1:90,1] + -52.301;
   1:  PR[GP1:91,2] = PR[GP1:90,2] + 10.823;
   1:L PR[91] R[100]mm/sec CNT100;
   1:  PR[GP1:91,1] = PR[GP1:90,1] + -54.308;
   1:  PR[GP1:91,2] = PR[GP1:90,2] + -0.082;
   1:L PR[91] R[100]mm/sec CNT100;
   1:  PR[GP1:91,1] = PR[GP1:90,1] + -54.041;
   1:  PR[GP1:91,2] = PR[GP1:90,2] + -1.866;
   1:L PR[91] R[100]mm/sec CNT100;
   1:  PR[GP1:91,1] = PR[GP1:90,1] + -51.617;
   1:  PR[GP1:91,2] = PR[GP1:90,2] + -15.006;
   1:L PR[91] R[100]mm/sec CNT100;
   1:  PR[GP1:91,1] = PR[GP1:90,1] + -50.808;
   1:  PR[GP1:91,2] = PR[GP1:90,2] + -16.373;
   1:L PR[91] R[100]mm/sec CNT100;
   1:  PR[GP1:91,1] = PR[GP1:90,1] + -43.675;
   1:  PR[GP1:91,2] = PR[GP1:90,2] + -28.171;
   1:L PR[91] R[100]mm/sec CNT100;
   1:  PR[GP1:91,1] = PR[GP1:90,1] + -42.755;
   1:  PR[GP1:91,2] = PR[GP1:90,2] + -28.930;
   1:L PR[91] R[100]mm/sec CNT100;
   1:  PR[GP1:91,1] = PR[GP1:90,1] + -31.441;
   1:  PR[GP1:91,2] = PR[GP1:90,2] + -37.885;
   1:L PR[91] R[100]mm/sec CNT100;
   1:  PR[GP1:91,1] = PR[GP1:90,1] + -30.846;
   1:  PR[GP1:91,2] = PR[GP1:90,2] + -38.104;
   1:L PR[91] R[100]mm/sec CNT100;
   1:  PR[GP1:91,1] = PR[GP1:90,1] + -16.394;
   1:  PR[GP1:91,2] = PR[GP1:90,2] + -42.845;
   1:L PR[91] R[100]mm/sec CNT100;
   1:  PR[GP1:91,1] = PR[GP1:90,1] + -14.454;
   1:  PR[GP1:91,2] = PR[GP1:90,2] + -42.781;
   1:L PR[91] R[100]mm/sec CNT100;
   1:  PR[GP1:91,1] = PR[GP1:90,1] + -0.852;
   1:  PR[GP1:91,2] = PR[GP1:90,2] + -42.426;
   1:L PR[91] R[100]mm/sec CNT100;
   1:  PR[GP1:91,1] = PR[GP1:90,1] + 1.068;
   1:  PR[GP1:91,2] = PR[GP1:90,2] + -42.427;
   1:L PR[91] R[100]mm/sec CNT100;
   1:  PR[GP1:91,1] = PR[GP1:90,1] + 14.665;
   1:  PR[GP1:91,2] = PR[GP1:90,2] + -42.780;
   1:L PR[91] R[100]mm/sec CNT100;
   1:  PR[GP1:91,1] = PR[GP1:90,1] + 16.610;
   1:  PR[GP1:91,2] = PR[GP1:90,2] + -42.845;
   1:L PR[91] R[100]mm/sec CNT100;
   1:  PR[GP1:91,1] = PR[GP1:90,1] + 31.061;
   1:  PR[GP1:91,2] = PR[GP1:90,2] + -38.104;
   1:L PR[91] R[100]mm/sec CNT100;
   1:  PR[GP1:91,1] = PR[GP1:90,1] + 31.656;
   1:  PR[GP1:91,2] = PR[GP1:90,2] + -37.885;
   1:L PR[91] R[100]mm/sec CNT100;
   1:  PR[GP1:91,1] = PR[GP1:90,1] + 42.969;
   1:  PR[GP1:91,2] = PR[GP1:90,2] + -28.928;
   1:L PR[91] R[100]mm/sec CNT100;
   1:  PR[GP1:91,1] = PR[GP1:90,1] + 43.889;
   1:  PR[GP1:91,2] = PR[GP1:90,2] + -28.168;
   1:L PR[91] R[100]mm/sec CNT100;
   1:  PR[GP1:91,1] = PR[GP1:90,1] + 51.022;
   1:  PR[GP1:91,2] = PR[GP1:90,2] + -16.376;
   1:L PR[91] R[100]mm/sec CNT100;
   1:  PR[GP1:91,1] = PR[GP1:90,1] + 51.830;
   1:  PR[GP1:91,2] = PR[GP1:90,2] + -15.013;
   1:L PR[91] R[100]mm/sec CNT100;
   1:  PR[GP1:91,1] = PR[GP1:90,1] + 52.132;
   1:  PR[GP1:91,2] = PR[GP1:90,2] + -13.343;
   1:L PR[91] R[100]mm/sec CNT100;
   1:  PR[GP1:91,1] = PR[GP1:90,1] + 52.514;
   1:  PR[GP1:91,2] = PR[GP1:90,2] + -10.970;
   1:L PR[91] R[100]mm/sec CNT100;
   1:  PR[GP1:91,1] = PR[GP1:90,1] + 54.521;
   1:  PR[GP1:91,2] = PR[GP1:90,2] + -0.062;
   1:L PR[91] R[100]mm/sec CNT100;
   1:  PR[GP1:91,1] = PR[GP1:90,1] + 54.254;
   1:  PR[GP1:91,2] = PR[GP1:90,2] + 1.724;
   1:L PR[91] R[100]mm/sec CNT100;
   1:  PR[GP1:91,1] = PR[GP1:90,1] + 51.830;
   1:  PR[GP1:91,2] = PR[GP1:90,2] + 14.869;
   1:L PR[91] R[100]mm/sec CNT100;
   1:  PR[GP1:91,1] = PR[GP1:90,1] + 51.023;
   1:  PR[GP1:91,2] = PR[GP1:90,2] + 16.232;
   1:L PR[91] R[100]mm/sec CNT100;
   1:  PR[GP1:91,1] = PR[GP1:90,1] + 43.889;
   1:  PR[GP1:91,2] = PR[GP1:90,2] + 28.025;
   1:L PR[91] R[100]mm/sec CNT100;
   1:  PR[GP1:91,1] = PR[GP1:90,1] + 42.969;
   1:  PR[GP1:91,2] = PR[GP1:90,2] + 28.785;
   1:L PR[91] R[100]mm/sec CNT100;
   1:  PR[GP1:91,1] = PR[GP1:90,1] + 31.654;
   1:  PR[GP1:91,2] = PR[GP1:90,2] + 37.742;
   1:L PR[91] R[100]mm/sec CNT100;
   1:  PR[GP1:91,1] = PR[GP1:90,1] + 31.059;
   1:  PR[GP1:91,2] = PR[GP1:90,2] + 37.961;
   1:L PR[91] R[100]mm/sec CNT100;
   1:  PR[GP1:91,1] = PR[GP1:90,1] + 16.606;
   1:  PR[GP1:91,2] = PR[GP1:90,2] + 42.701;
   1:L PR[91] R[100]mm/sec CNT100;
   1:  PR[GP1:91,1] = PR[GP1:90,1] + 14.694;
   1:  PR[GP1:91,2] = PR[GP1:90,2] + 42.638;
   1:L PR[91] R[100]mm/sec CNT100;
   1:  PR[GP1:91,1] = PR[GP1:90,1] + 1.068;
   1:  PR[GP1:91,2] = PR[GP1:90,2] + 42.282;
   1:L PR[91] R[100]mm/sec CNT100;
   1:  ! -- Layer/Ebene 166 -- !;
   1:  PR[91] = PR[90];
   1:  PR[GP1:91,1] = PR[GP1:90,1] + -0.829;
   1:  PR[GP1:91,2] = PR[GP1:90,2] + 42.442;
   1:  PR[GP1:91,3] = PR[GP1:90,3] + 101.565;
   1:L PR[91] R[100]mm/sec CNT100;
   1:  PR[GP1:91,1] = PR[GP1:90,1] + -16.110;
   1:  PR[GP1:91,2] = PR[GP1:90,2] + 42.839;
   1:L PR[91] R[100]mm/sec CNT100;
   1:  PR[GP1:91,1] = PR[GP1:90,1] + -16.194;
   1:  PR[GP1:91,2] = PR[GP1:90,2] + 42.828;
   1:L PR[91] R[100]mm/sec CNT100;
   1:  PR[GP1:91,1] = PR[GP1:90,1] + -21.100;
   1:  PR[GP1:91,2] = PR[GP1:90,2] + 41.177;
   1:L PR[91] R[100]mm/sec CNT100;
   1:  PR[GP1:91,1] = PR[GP1:90,1] + -30.912;
   1:  PR[GP1:91,2] = PR[GP1:90,2] + 37.959;
   1:L PR[91] R[100]mm/sec CNT100;
   1:  PR[GP1:91,1] = PR[GP1:90,1] + -31.217;
   1:  PR[GP1:91,2] = PR[GP1:90,2] + 37.847;
   1:L PR[91] R[100]mm/sec CNT100;
   1:  PR[GP1:91,1] = PR[GP1:90,1] + -42.815;
   1:  PR[GP1:91,2] = PR[GP1:90,2] + 28.669;
   1:L PR[91] R[100]mm/sec CNT100;
   1:  PR[GP1:91,1] = PR[GP1:90,1] + -43.490;
   1:  PR[GP1:91,2] = PR[GP1:90,2] + 28.112;
   1:L PR[91] R[100]mm/sec CNT100;
   1:  PR[GP1:91,1] = PR[GP1:90,1] + -50.816;
   1:  PR[GP1:91,2] = PR[GP1:90,2] + 15.996;
   1:L PR[91] R[100]mm/sec CNT100;
   1:  PR[GP1:91,1] = PR[GP1:90,1] + -51.457;
   1:  PR[GP1:91,2] = PR[GP1:90,2] + 14.910;
   1:L PR[91] R[100]mm/sec CNT100;
   1:  PR[GP1:91,1] = PR[GP1:90,1] + -51.698;
   1:  PR[GP1:91,2] = PR[GP1:90,2] + 13.584;
   1:L PR[91] R[100]mm/sec CNT100;
   1:  PR[GP1:91,1] = PR[GP1:90,1] + -52.007;
   1:  PR[GP1:91,2] = PR[GP1:90,2] + 11.666;
   1:L PR[91] R[100]mm/sec CNT100;
   1:  PR[GP1:91,1] = PR[GP1:90,1] + -54.170;
   1:  PR[GP1:91,2] = PR[GP1:90,2] + -0.082;
   1:L PR[91] R[100]mm/sec CNT100;
   1:  PR[GP1:91,1] = PR[GP1:90,1] + -53.951;
   1:  PR[GP1:91,2] = PR[GP1:90,2] + -1.540;
   1:L PR[91] R[100]mm/sec CNT100;
   1:  PR[GP1:91,1] = PR[GP1:90,1] + -51.458;
   1:  PR[GP1:91,2] = PR[GP1:90,2] + -15.053;
   1:L PR[91] R[100]mm/sec CNT100;
   1:  PR[GP1:91,1] = PR[GP1:90,1] + -50.815;
   1:  PR[GP1:91,2] = PR[GP1:90,2] + -16.140;
   1:L PR[91] R[100]mm/sec CNT100;
   1:  PR[GP1:91,1] = PR[GP1:90,1] + -43.491;
   1:  PR[GP1:91,2] = PR[GP1:90,2] + -28.255;
   1:L PR[91] R[100]mm/sec CNT100;
   1:  PR[GP1:91,1] = PR[GP1:90,1] + -42.815;
   1:  PR[GP1:91,2] = PR[GP1:90,2] + -28.812;
   1:L PR[91] R[100]mm/sec CNT100;
   1:  PR[GP1:91,1] = PR[GP1:90,1] + -31.220;
   1:  PR[GP1:91,2] = PR[GP1:90,2] + -37.990;
   1:L PR[91] R[100]mm/sec CNT100;
   1:  PR[GP1:91,1] = PR[GP1:90,1] + -30.915;
   1:  PR[GP1:91,2] = PR[GP1:90,2] + -38.102;
   1:L PR[91] R[100]mm/sec CNT100;
   1:  PR[GP1:91,1] = PR[GP1:90,1] + -21.100;
   1:  PR[GP1:91,2] = PR[GP1:90,2] + -41.322;
   1:L PR[91] R[100]mm/sec CNT100;
   1:  PR[GP1:91,1] = PR[GP1:90,1] + -16.198;
   1:  PR[GP1:91,2] = PR[GP1:90,2] + -42.972;
   1:L PR[91] R[100]mm/sec CNT100;
   1:  PR[GP1:91,1] = PR[GP1:90,1] + -16.114;
   1:  PR[GP1:91,2] = PR[GP1:90,2] + -42.982;
   1:L PR[91] R[100]mm/sec CNT100;
   1:  PR[GP1:91,1] = PR[GP1:90,1] + -0.829;
   1:  PR[GP1:91,2] = PR[GP1:90,2] + -42.586;
   1:L PR[91] R[100]mm/sec CNT100;
   1:  PR[GP1:91,1] = PR[GP1:90,1] + 1.045;
   1:L PR[91] R[100]mm/sec CNT100;
   1:  PR[GP1:91,1] = PR[GP1:90,1] + 16.045;
   1:  PR[GP1:91,2] = PR[GP1:90,2] + -42.976;
   1:L PR[91] R[100]mm/sec CNT100;
   1:  PR[GP1:91,1] = PR[GP1:90,1] + 16.329;
   1:  PR[GP1:91,2] = PR[GP1:90,2] + -42.982;
   1:L PR[91] R[100]mm/sec CNT100;
   1:  PR[GP1:91,1] = PR[GP1:90,1] + 16.414;
   1:  PR[GP1:91,2] = PR[GP1:90,2] + -42.972;
   1:L PR[91] R[100]mm/sec CNT100;
   1:  PR[GP1:91,1] = PR[GP1:90,1] + 21.310;
   1:  PR[GP1:91,2] = PR[GP1:90,2] + -41.323;
   1:L PR[91] R[100]mm/sec CNT100;
   1:  PR[GP1:91,1] = PR[GP1:90,1] + 31.130;
   1:  PR[GP1:91,2] = PR[GP1:90,2] + -38.102;
   1:L PR[91] R[100]mm/sec CNT100;
   1:  PR[GP1:91,1] = PR[GP1:90,1] + 31.435;
   1:  PR[GP1:91,2] = PR[GP1:90,2] + -37.989;
   1:L PR[91] R[100]mm/sec CNT100;
   1:  PR[GP1:91,1] = PR[GP1:90,1] + 43.029;
   1:  PR[GP1:91,2] = PR[GP1:90,2] + -28.810;
   1:L PR[91] R[100]mm/sec CNT100;
   1:  PR[GP1:91,1] = PR[GP1:90,1] + 43.705;
   1:  PR[GP1:91,2] = PR[GP1:90,2] + -28.252;
   1:L PR[91] R[100]mm/sec CNT100;
   1:  PR[GP1:91,1] = PR[GP1:90,1] + 51.029;
   1:  PR[GP1:91,2] = PR[GP1:90,2] + -16.143;
   1:L PR[91] R[100]mm/sec CNT100;
   1:  PR[GP1:91,1] = PR[GP1:90,1] + 51.671;
   1:  PR[GP1:91,2] = PR[GP1:90,2] + -15.060;
   1:L PR[91] R[100]mm/sec CNT100;
   1:  PR[GP1:91,1] = PR[GP1:90,1] + 51.912;
   1:  PR[GP1:91,2] = PR[GP1:90,2] + -13.731;
   1:L PR[91] R[100]mm/sec CNT100;
   1:  PR[GP1:91,1] = PR[GP1:90,1] + 52.221;
   1:  PR[GP1:91,2] = PR[GP1:90,2] + -11.812;
   1:L PR[91] R[100]mm/sec CNT100;
   1:  PR[GP1:91,1] = PR[GP1:90,1] + 54.383;
   1:  PR[GP1:91,2] = PR[GP1:90,2] + -0.062;
   1:L PR[91] R[100]mm/sec CNT100;
   1:  PR[GP1:91,1] = PR[GP1:90,1] + 54.165;
   1:  PR[GP1:91,2] = PR[GP1:90,2] + 1.398;
   1:L PR[91] R[100]mm/sec CNT100;
   1:  PR[GP1:91,1] = PR[GP1:90,1] + 51.671;
   1:  PR[GP1:91,2] = PR[GP1:90,2] + 14.916;
   1:L PR[91] R[100]mm/sec CNT100;
   1:  PR[GP1:91,1] = PR[GP1:90,1] + 51.029;
   1:  PR[GP1:91,2] = PR[GP1:90,2] + 16.000;
   1:L PR[91] R[100]mm/sec CNT100;
   1:  PR[GP1:91,1] = PR[GP1:90,1] + 43.704;
   1:  PR[GP1:91,2] = PR[GP1:90,2] + 28.109;
   1:L PR[91] R[100]mm/sec CNT100;
   1:  PR[GP1:91,1] = PR[GP1:90,1] + 43.029;
   1:  PR[GP1:91,2] = PR[GP1:90,2] + 28.667;
   1:L PR[91] R[100]mm/sec CNT100;
   1:  PR[GP1:91,1] = PR[GP1:90,1] + 31.432;
   1:  PR[GP1:91,2] = PR[GP1:90,2] + 37.847;
   1:L PR[91] R[100]mm/sec CNT100;
   1:  PR[GP1:91,1] = PR[GP1:90,1] + 31.128;
   1:  PR[GP1:91,2] = PR[GP1:90,2] + 37.959;
   1:L PR[91] R[100]mm/sec CNT100;
   1:  PR[GP1:91,1] = PR[GP1:90,1] + 21.311;
   1:  PR[GP1:91,2] = PR[GP1:90,2] + 41.179;
   1:L PR[91] R[100]mm/sec CNT100;
   1:  PR[GP1:91,1] = PR[GP1:90,1] + 16.410;
   1:  PR[GP1:91,2] = PR[GP1:90,2] + 42.828;
   1:L PR[91] R[100]mm/sec CNT100;
   1:  PR[GP1:91,1] = PR[GP1:90,1] + 16.326;
   1:  PR[GP1:91,2] = PR[GP1:90,2] + 42.839;
   1:L PR[91] R[100]mm/sec CNT100;
   1:  PR[GP1:91,1] = PR[GP1:90,1] + 1.045;
   1:  PR[GP1:91,2] = PR[GP1:90,2] + 42.442;
   1:L PR[91] R[100]mm/sec CNT100;
   1:  ! -- Layer/Ebene 167 -- !;
   1:  PR[91] = PR[90];
   1:  PR[GP1:91,1] = PR[GP1:90,1] + -0.807;
   1:  PR[GP1:91,2] = PR[GP1:90,2] + 42.601;
   1:  PR[GP1:91,3] = PR[GP1:90,3] + 102.175;
   1:L PR[91] R[100]mm/sec CNT100;
   1:  PR[GP1:91,1] = PR[GP1:90,1] + -15.739;
   1:  PR[GP1:91,2] = PR[GP1:90,2] + 42.987;
   1:L PR[91] R[100]mm/sec CNT100;
   1:  PR[GP1:91,1] = PR[GP1:90,1] + -16.097;
   1:  PR[GP1:91,2] = PR[GP1:90,2] + 42.942;
   1:L PR[91] R[100]mm/sec CNT100;
   1:  PR[GP1:91,1] = PR[GP1:90,1] + -28.209;
   1:  PR[GP1:91,2] = PR[GP1:90,2] + 38.867;
   1:L PR[91] R[100]mm/sec CNT100;
   1:  PR[GP1:91,1] = PR[GP1:90,1] + -31.004;
   1:  PR[GP1:91,2] = PR[GP1:90,2] + 37.945;
   1:L PR[91] R[100]mm/sec CNT100;
   1:  PR[GP1:91,1] = PR[GP1:90,1] + -42.875;
   1:  PR[GP1:91,2] = PR[GP1:90,2] + 28.552;
   1:L PR[91] R[100]mm/sec CNT100;
   1:  PR[GP1:91,1] = PR[GP1:90,1] + -43.305;
   1:  PR[GP1:91,2] = PR[GP1:90,2] + 28.197;
   1:L PR[91] R[100]mm/sec CNT100;
   1:  PR[GP1:91,1] = PR[GP1:90,1] + -51.300;
   1:  PR[GP1:91,2] = PR[GP1:90,2] + 14.955;
   1:L PR[91] R[100]mm/sec CNT100;
   1:  PR[GP1:91,1] = PR[GP1:90,1] + -51.478;
   1:  PR[GP1:91,2] = PR[GP1:90,2] + 13.972;
   1:L PR[91] R[100]mm/sec CNT100;
   1:  PR[GP1:91,1] = PR[GP1:90,1] + -51.714;
   1:  PR[GP1:91,2] = PR[GP1:90,2] + 12.508;
   1:L PR[91] R[100]mm/sec CNT100;
   1:  PR[GP1:91,1] = PR[GP1:90,1] + -54.031;
   1:  PR[GP1:91,2] = PR[GP1:90,2] + -0.082;
   1:L PR[91] R[100]mm/sec CNT100;
   1:  PR[GP1:91,1] = PR[GP1:90,1] + -53.862;
   1:  PR[GP1:91,2] = PR[GP1:90,2] + -1.215;
   1:L PR[91] R[100]mm/sec CNT100;
   1:  PR[GP1:91,1] = PR[GP1:90,1] + -51.300;
   1:  PR[GP1:91,2] = PR[GP1:90,2] + -15.097;
   1:L PR[91] R[100]mm/sec CNT100;
   1:  PR[GP1:91,1] = PR[GP1:90,1] + -43.306;
   1:  PR[GP1:91,2] = PR[GP1:90,2] + -28.339;
   1:L PR[91] R[100]mm/sec CNT100;
   1:  PR[GP1:91,1] = PR[GP1:90,1] + -42.876;
   1:  PR[GP1:91,2] = PR[GP1:90,2] + -28.694;
   1:L PR[91] R[100]mm/sec CNT100;
   1:  PR[GP1:91,1] = PR[GP1:90,1] + -31.007;
   1:  PR[GP1:91,2] = PR[GP1:90,2] + -38.088;
   1:L PR[91] R[100]mm/sec CNT100;
   1:  PR[GP1:91,1] = PR[GP1:90,1] + -28.208;
   1:  PR[GP1:91,2] = PR[GP1:90,2] + -39.010;
   1:L PR[91] R[100]mm/sec CNT100;
   1:  PR[GP1:91,1] = PR[GP1:90,1] + -16.101;
   1:  PR[GP1:91,2] = PR[GP1:90,2] + -43.086;
   1:L PR[91] R[100]mm/sec CNT100;
   1:  PR[GP1:91,1] = PR[GP1:90,1] + -15.744;
   1:  PR[GP1:91,2] = PR[GP1:90,2] + -43.130;
   1:L PR[91] R[100]mm/sec CNT100;
   1:  PR[GP1:91,1] = PR[GP1:90,1] + -0.807;
   1:  PR[GP1:91,2] = PR[GP1:90,2] + -42.745;
   1:L PR[91] R[100]mm/sec CNT100;
   1:  PR[GP1:91,1] = PR[GP1:90,1] + 1.022;
   1:L PR[91] R[100]mm/sec CNT100;
   1:  PR[GP1:91,1] = PR[GP1:90,1] + 15.959;
   1:  PR[GP1:91,2] = PR[GP1:90,2] + -43.130;
   1:L PR[91] R[100]mm/sec CNT100;
   1:  PR[GP1:91,1] = PR[GP1:90,1] + 16.317;
   1:  PR[GP1:91,2] = PR[GP1:90,2] + -43.086;
   1:L PR[91] R[100]mm/sec CNT100;
   1:  PR[GP1:91,1] = PR[GP1:90,1] + 28.419;
   1:  PR[GP1:91,2] = PR[GP1:90,2] + -39.012;
   1:L PR[91] R[100]mm/sec CNT100;
   1:  PR[GP1:91,1] = PR[GP1:90,1] + 31.222;
   1:  PR[GP1:91,2] = PR[GP1:90,2] + -38.087;
   1:L PR[91] R[100]mm/sec CNT100;
   1:  PR[GP1:91,1] = PR[GP1:90,1] + 43.089;
   1:  PR[GP1:91,2] = PR[GP1:90,2] + -28.692;
   1:L PR[91] R[100]mm/sec CNT100;
   1:  PR[GP1:91,1] = PR[GP1:90,1] + 43.520;
   1:  PR[GP1:91,2] = PR[GP1:90,2] + -28.336;
   1:L PR[91] R[100]mm/sec CNT100;
   1:  PR[GP1:91,1] = PR[GP1:90,1] + 51.513;
   1:  PR[GP1:91,2] = PR[GP1:90,2] + -15.104;
   1:L PR[91] R[100]mm/sec CNT100;
   1:  PR[GP1:91,1] = PR[GP1:90,1] + 51.692;
   1:  PR[GP1:91,2] = PR[GP1:90,2] + -14.119;
   1:L PR[91] R[100]mm/sec CNT100;
   1:  PR[GP1:91,1] = PR[GP1:90,1] + 51.927;
   1:  PR[GP1:91,2] = PR[GP1:90,2] + -12.655;
   1:L PR[91] R[100]mm/sec CNT100;
   1:  PR[GP1:91,1] = PR[GP1:90,1] + 54.245;
   1:  PR[GP1:91,2] = PR[GP1:90,2] + -0.062;
   1:L PR[91] R[100]mm/sec CNT100;
   1:  PR[GP1:91,1] = PR[GP1:90,1] + 54.075;
   1:  PR[GP1:91,2] = PR[GP1:90,2] + 1.072;
   1:L PR[91] R[100]mm/sec CNT100;
   1:  PR[GP1:91,1] = PR[GP1:90,1] + 51.513;
   1:  PR[GP1:91,2] = PR[GP1:90,2] + 14.960;
   1:L PR[91] R[100]mm/sec CNT100;
   1:  PR[GP1:91,1] = PR[GP1:90,1] + 43.519;
   1:  PR[GP1:91,2] = PR[GP1:90,2] + 28.193;
   1:L PR[91] R[100]mm/sec CNT100;
   1:  PR[GP1:91,1] = PR[GP1:90,1] + 43.089;
   1:  PR[GP1:91,2] = PR[GP1:90,2] + 28.549;
   1:L PR[91] R[100]mm/sec CNT100;
   1:  PR[GP1:91,1] = PR[GP1:90,1] + 31.219;
   1:  PR[GP1:91,2] = PR[GP1:90,2] + 37.945;
   1:L PR[91] R[100]mm/sec CNT100;
   1:  PR[GP1:91,1] = PR[GP1:90,1] + 28.420;
   1:  PR[GP1:91,2] = PR[GP1:90,2] + 38.867;
   1:L PR[91] R[100]mm/sec CNT100;
   1:  PR[GP1:91,1] = PR[GP1:90,1] + 16.313;
   1:  PR[GP1:91,2] = PR[GP1:90,2] + 42.942;
   1:L PR[91] R[100]mm/sec CNT100;
   1:  PR[GP1:91,1] = PR[GP1:90,1] + 15.955;
   1:  PR[GP1:91,2] = PR[GP1:90,2] + 42.987;
   1:L PR[91] R[100]mm/sec CNT100;
   1:  PR[GP1:91,1] = PR[GP1:90,1] + 1.022;
   1:  PR[GP1:91,2] = PR[GP1:90,2] + 42.601;
   1:L PR[91] R[100]mm/sec CNT100;
   1:  ! -- Layer/Ebene 168 -- !;
   1:  PR[91] = PR[90];
   1:  PR[GP1:91,1] = PR[GP1:90,1] + -0.784;
   1:  PR[GP1:91,2] = PR[GP1:90,2] + 42.760;
   1:  PR[GP1:91,3] = PR[GP1:90,3] + 102.785;
   1:L PR[91] R[100]mm/sec CNT100;
   1:  PR[GP1:91,1] = PR[GP1:90,1] + -15.369;
   1:  PR[GP1:91,2] = PR[GP1:90,2] + 43.135;
   1:L PR[91] R[100]mm/sec CNT100;
   1:  PR[GP1:91,1] = PR[GP1:90,1] + -16.001;
   1:  PR[GP1:91,2] = PR[GP1:90,2] + 43.057;
   1:L PR[91] R[100]mm/sec CNT100;
   1:  PR[GP1:91,1] = PR[GP1:90,1] + -30.804;
   1:  PR[GP1:91,2] = PR[GP1:90,2] + 38.066;
   1:L PR[91] R[100]mm/sec CNT100;
   1:  PR[GP1:91,1] = PR[GP1:90,1] + -35.147;
   1:  PR[GP1:91,2] = PR[GP1:90,2] + 34.597;
   1:L PR[91] R[100]mm/sec CNT100;
   1:  PR[GP1:91,1] = PR[GP1:90,1] + -43.124;
   1:  PR[GP1:91,2] = PR[GP1:90,2] + 28.275;
   1:L PR[91] R[100]mm/sec CNT100;
   1:  PR[GP1:91,1] = PR[GP1:90,1] + -51.139;
   1:  PR[GP1:91,2] = PR[GP1:90,2] + 15.005;
   1:L PR[91] R[100]mm/sec CNT100;
   1:  PR[GP1:91,1] = PR[GP1:90,1] + -51.421;
   1:  PR[GP1:91,2] = PR[GP1:90,2] + 13.348;
   1:L PR[91] R[100]mm/sec CNT100;
   1:  PR[GP1:91,1] = PR[GP1:90,1] + -53.893;
   1:  PR[GP1:91,2] = PR[GP1:90,2] + -0.082;
   1:L PR[91] R[100]mm/sec CNT100;
   1:  PR[GP1:91,1] = PR[GP1:90,1] + -53.772;
   1:  PR[GP1:91,2] = PR[GP1:90,2] + -0.889;
   1:L PR[91] R[100]mm/sec CNT100;
   1:  PR[GP1:91,1] = PR[GP1:90,1] + -51.142;
   1:  PR[GP1:91,2] = PR[GP1:90,2] + -15.144;
   1:L PR[91] R[100]mm/sec CNT100;
   1:  PR[GP1:91,1] = PR[GP1:90,1] + -43.125;
   1:  PR[GP1:91,2] = PR[GP1:90,2] + -28.418;
   1:L PR[91] R[100]mm/sec CNT100;
   1:  PR[GP1:91,1] = PR[GP1:90,1] + -35.146;
   1:  PR[GP1:91,2] = PR[GP1:90,2] + -34.742;
   1:L PR[91] R[100]mm/sec CNT100;
   1:  PR[GP1:91,1] = PR[GP1:90,1] + -30.881;
   1:  PR[GP1:91,2] = PR[GP1:90,2] + -38.163;
   1:L PR[91] R[100]mm/sec CNT100;
   1:  PR[GP1:91,1] = PR[GP1:90,1] + -30.824;
   1:  PR[GP1:91,2] = PR[GP1:90,2] + -38.203;
   1:L PR[91] R[100]mm/sec CNT100;
   1:  PR[GP1:91,1] = PR[GP1:90,1] + -16.005;
   1:  PR[GP1:91,2] = PR[GP1:90,2] + -43.200;
   1:L PR[91] R[100]mm/sec CNT100;
   1:  PR[GP1:91,1] = PR[GP1:90,1] + -15.373;
   1:  PR[GP1:91,2] = PR[GP1:90,2] + -43.278;
   1:L PR[91] R[100]mm/sec CNT100;
   1:  PR[GP1:91,1] = PR[GP1:90,1] + -0.784;
   1:  PR[GP1:91,2] = PR[GP1:90,2] + -42.904;
   1:L PR[91] R[100]mm/sec CNT100;
   1:  PR[GP1:91,1] = PR[GP1:90,1] + 0.999;
   1:L PR[91] R[100]mm/sec CNT100;
   1:  PR[GP1:91,1] = PR[GP1:90,1] + 15.589;
   1:  PR[GP1:91,2] = PR[GP1:90,2] + -43.278;
   1:L PR[91] R[100]mm/sec CNT100;
   1:  PR[GP1:91,1] = PR[GP1:90,1] + 16.220;
   1:  PR[GP1:91,2] = PR[GP1:90,2] + -43.200;
   1:L PR[91] R[100]mm/sec CNT100;
   1:  PR[GP1:91,1] = PR[GP1:90,1] + 31.022;
   1:  PR[GP1:91,2] = PR[GP1:90,2] + -38.208;
   1:L PR[91] R[100]mm/sec CNT100;
   1:  PR[GP1:91,1] = PR[GP1:90,1] + 35.357;
   1:  PR[GP1:91,2] = PR[GP1:90,2] + -34.743;
   1:L PR[91] R[100]mm/sec CNT100;
   1:  PR[GP1:91,1] = PR[GP1:90,1] + 43.339;
   1:  PR[GP1:91,2] = PR[GP1:90,2] + -28.415;
   1:L PR[91] R[100]mm/sec CNT100;
   1:  PR[GP1:91,1] = PR[GP1:90,1] + 51.353;
   1:  PR[GP1:91,2] = PR[GP1:90,2] + -15.154;
   1:L PR[91] R[100]mm/sec CNT100;
   1:  PR[GP1:91,1] = PR[GP1:90,1] + 51.634;
   1:  PR[GP1:91,2] = PR[GP1:90,2] + -13.496;
   1:L PR[91] R[100]mm/sec CNT100;
   1:  PR[GP1:91,1] = PR[GP1:90,1] + 54.106;
   1:  PR[GP1:91,2] = PR[GP1:90,2] + -0.062;
   1:L PR[91] R[100]mm/sec CNT100;
   1:  PR[GP1:91,1] = PR[GP1:90,1] + 53.985;
   1:  PR[GP1:91,2] = PR[GP1:90,2] + 0.746;
   1:L PR[91] R[100]mm/sec CNT100;
   1:  PR[GP1:91,1] = PR[GP1:90,1] + 51.355;
   1:  PR[GP1:91,2] = PR[GP1:90,2] + 15.007;
   1:L PR[91] R[100]mm/sec CNT100;
   1:  PR[GP1:91,1] = PR[GP1:90,1] + 43.338;
   1:  PR[GP1:91,2] = PR[GP1:90,2] + 28.272;
   1:L PR[91] R[100]mm/sec CNT100;
   1:  PR[GP1:91,1] = PR[GP1:90,1] + 35.357;
   1:  PR[GP1:91,2] = PR[GP1:90,2] + 34.599;
   1:L PR[91] R[100]mm/sec CNT100;
   1:  PR[GP1:91,1] = PR[GP1:90,1] + 31.093;
   1:  PR[GP1:91,2] = PR[GP1:90,2] + 38.020;
   1:L PR[91] R[100]mm/sec CNT100;
   1:  PR[GP1:91,1] = PR[GP1:90,1] + 31.037;
   1:  PR[GP1:91,2] = PR[GP1:90,2] + 38.060;
   1:L PR[91] R[100]mm/sec CNT100;
   1:  PR[GP1:91,1] = PR[GP1:90,1] + 16.216;
   1:  PR[GP1:91,2] = PR[GP1:90,2] + 43.056;
   1:L PR[91] R[100]mm/sec CNT100;
   1:  PR[GP1:91,1] = PR[GP1:90,1] + 15.585;
   1:  PR[GP1:91,2] = PR[GP1:90,2] + 43.135;
   1:L PR[91] R[100]mm/sec CNT100;
   1:  PR[GP1:91,1] = PR[GP1:90,1] + 1.000;
   1:  PR[GP1:91,2] = PR[GP1:90,2] + 42.760;
   1:L PR[91] R[100]mm/sec CNT100;
   1:  ! -- Layer/Ebene 169 -- !;
   1:  PR[91] = PR[90];
   1:  PR[GP1:91,1] = PR[GP1:90,1] + -0.762;
   1:  PR[GP1:91,2] = PR[GP1:90,2] + 42.919;
   1:  PR[GP1:91,3] = PR[GP1:90,3] + 103.395;
   1:L PR[91] R[100]mm/sec CNT100;
   1:  PR[GP1:91,1] = PR[GP1:90,1] + -14.998;
   1:  PR[GP1:91,2] = PR[GP1:90,2] + 43.283;
   1:L PR[91] R[100]mm/sec CNT100;
   1:  PR[GP1:91,1] = PR[GP1:90,1] + -15.904;
   1:  PR[GP1:91,2] = PR[GP1:90,2] + 43.171;
   1:L PR[91] R[100]mm/sec CNT100;
   1:  PR[GP1:91,1] = PR[GP1:90,1] + -30.278;
   1:  PR[GP1:91,2] = PR[GP1:90,2] + 38.333;
   1:L PR[91] R[100]mm/sec CNT100;
   1:  PR[GP1:91,1] = PR[GP1:90,1] + -30.614;
   1:  PR[GP1:91,2] = PR[GP1:90,2] + 38.203;
   1:L PR[91] R[100]mm/sec CNT100;
   1:  PR[GP1:91,1] = PR[GP1:90,1] + -42.938;
   1:  PR[GP1:91,2] = PR[GP1:90,2] + 28.360;
   1:L PR[91] R[100]mm/sec CNT100;
   1:  PR[GP1:91,1] = PR[GP1:90,1] + -50.981;
   1:  PR[GP1:91,2] = PR[GP1:90,2] + 15.052;
   1:L PR[91] R[100]mm/sec CNT100;
   1:  PR[GP1:91,1] = PR[GP1:90,1] + -51.127;
   1:  PR[GP1:91,2] = PR[GP1:90,2] + 14.191;
   1:L PR[91] R[100]mm/sec CNT100;
   1:  PR[GP1:91,1] = PR[GP1:90,1] + -53.754;
   1:  PR[GP1:91,2] = PR[GP1:90,2] + -0.082;
   1:L PR[91] R[100]mm/sec CNT100;
   1:  PR[GP1:91,1] = PR[GP1:90,1] + -53.682;
   1:  PR[GP1:91,2] = PR[GP1:90,2] + -0.563;
   1:L PR[91] R[100]mm/sec CNT100;
   1:  PR[GP1:91,1] = PR[GP1:90,1] + -50.983;
   1:  PR[GP1:91,2] = PR[GP1:90,2] + -15.191;
   1:L PR[91] R[100]mm/sec CNT100;
   1:  PR[GP1:91,1] = PR[GP1:90,1] + -42.940;
   1:  PR[GP1:91,2] = PR[GP1:90,2] + -28.503;
   1:L PR[91] R[100]mm/sec CNT100;
   1:  PR[GP1:91,1] = PR[GP1:90,1] + -30.937;
   1:  PR[GP1:91,2] = PR[GP1:90,2] + -38.124;
   1:L PR[91] R[100]mm/sec CNT100;
   1:  PR[GP1:91,1] = PR[GP1:90,1] + -30.633;
   1:  PR[GP1:91,2] = PR[GP1:90,2] + -38.339;
   1:L PR[91] R[100]mm/sec CNT100;
   1:  PR[GP1:91,1] = PR[GP1:90,1] + -30.281;
   1:  PR[GP1:91,2] = PR[GP1:90,2] + -38.476;
   1:L PR[91] R[100]mm/sec CNT100;
   1:  PR[GP1:91,1] = PR[GP1:90,1] + -15.908;
   1:  PR[GP1:91,2] = PR[GP1:90,2] + -43.314;
   1:L PR[91] R[100]mm/sec CNT100;
   1:  PR[GP1:91,1] = PR[GP1:90,1] + -15.002;
   1:  PR[GP1:91,2] = PR[GP1:90,2] + -43.426;
   1:L PR[91] R[100]mm/sec CNT100;
   1:  PR[GP1:91,1] = PR[GP1:90,1] + -0.761;
   1:  PR[GP1:91,2] = PR[GP1:90,2] + -43.064;
   1:L PR[91] R[100]mm/sec CNT100;
   1:  PR[GP1:91,1] = PR[GP1:90,1] + 0.977;
   1:L PR[91] R[100]mm/sec CNT100;
   1:  PR[GP1:91,1] = PR[GP1:90,1] + 15.218;
   1:  PR[GP1:91,2] = PR[GP1:90,2] + -43.426;
   1:L PR[91] R[100]mm/sec CNT100;
   1:  PR[GP1:91,1] = PR[GP1:90,1] + 16.124;
   1:  PR[GP1:91,2] = PR[GP1:90,2] + -43.314;
   1:L PR[91] R[100]mm/sec CNT100;
   1:  PR[GP1:91,1] = PR[GP1:90,1] + 30.496;
   1:  PR[GP1:91,2] = PR[GP1:90,2] + -38.475;
   1:L PR[91] R[100]mm/sec CNT100;
   1:  PR[GP1:91,1] = PR[GP1:90,1] + 30.831;
   1:  PR[GP1:91,2] = PR[GP1:90,2] + -38.345;
   1:L PR[91] R[100]mm/sec CNT100;
   1:  PR[GP1:91,1] = PR[GP1:90,1] + 43.154;
   1:  PR[GP1:91,2] = PR[GP1:90,2] + -28.500;
   1:L PR[91] R[100]mm/sec CNT100;
   1:  PR[GP1:91,1] = PR[GP1:90,1] + 51.195;
   1:  PR[GP1:91,2] = PR[GP1:90,2] + -15.200;
   1:L PR[91] R[100]mm/sec CNT100;
   1:  PR[GP1:91,1] = PR[GP1:90,1] + 51.341;
   1:  PR[GP1:91,2] = PR[GP1:90,2] + -14.338;
   1:L PR[91] R[100]mm/sec CNT100;
   1:  PR[GP1:91,1] = PR[GP1:90,1] + 53.968;
   1:  PR[GP1:91,2] = PR[GP1:90,2] + -0.062;
   1:L PR[91] R[100]mm/sec CNT100;
   1:  PR[GP1:91,1] = PR[GP1:90,1] + 53.896;
   1:  PR[GP1:91,2] = PR[GP1:90,2] + 0.420;
   1:L PR[91] R[100]mm/sec CNT100;
   1:  PR[GP1:91,1] = PR[GP1:90,1] + 51.196;
   1:  PR[GP1:91,2] = PR[GP1:90,2] + 15.056;
   1:L PR[91] R[100]mm/sec CNT100;
   1:  PR[GP1:91,1] = PR[GP1:90,1] + 51.050;
   1:  PR[GP1:91,2] = PR[GP1:90,2] + 15.302;
   1:L PR[91] R[100]mm/sec CNT100;
   1:  PR[GP1:91,1] = PR[GP1:90,1] + 43.153;
   1:  PR[GP1:91,2] = PR[GP1:90,2] + 28.358;
   1:L PR[91] R[100]mm/sec CNT100;
   1:  PR[GP1:91,1] = PR[GP1:90,1] + 31.149;
   1:  PR[GP1:91,2] = PR[GP1:90,2] + 37.981;
   1:L PR[91] R[100]mm/sec CNT100;
   1:  PR[GP1:91,1] = PR[GP1:90,1] + 30.845;
   1:  PR[GP1:91,2] = PR[GP1:90,2] + 38.196;
   1:L PR[91] R[100]mm/sec CNT100;
   1:  PR[GP1:91,1] = PR[GP1:90,1] + 30.494;
   1:  PR[GP1:91,2] = PR[GP1:90,2] + 38.332;
   1:L PR[91] R[100]mm/sec CNT100;
   1:  PR[GP1:91,1] = PR[GP1:90,1] + 16.120;
   1:  PR[GP1:91,2] = PR[GP1:90,2] + 43.170;
   1:L PR[91] R[100]mm/sec CNT100;
   1:  PR[GP1:91,1] = PR[GP1:90,1] + 15.214;
   1:  PR[GP1:91,2] = PR[GP1:90,2] + 43.283;
   1:L PR[91] R[100]mm/sec CNT100;
   1:  PR[GP1:91,1] = PR[GP1:90,1] + 0.977;
   1:  PR[GP1:91,2] = PR[GP1:90,2] + 42.920;
   1:L PR[91] R[100]mm/sec CNT100;
   1:  ! -- Layer/Ebene 170 -- !;
   1:  PR[91] = PR[90];
   1:  PR[GP1:91,1] = PR[GP1:90,1] + -0.739;
   1:  PR[GP1:91,2] = PR[GP1:90,2] + 43.079;
   1:  PR[GP1:91,3] = PR[GP1:90,3] + 104.005;
   1:L PR[91] R[100]mm/sec CNT100;
   1:  PR[GP1:91,1] = PR[GP1:90,1] + -14.628;
   1:  PR[GP1:91,2] = PR[GP1:90,2] + 43.431;
   1:L PR[91] R[100]mm/sec CNT100;
   1:  PR[GP1:91,1] = PR[GP1:90,1] + -15.808;
   1:  PR[GP1:91,2] = PR[GP1:90,2] + 43.285;
   1:L PR[91] R[100]mm/sec CNT100;
   1:  PR[GP1:91,1] = PR[GP1:90,1] + -29.828;
   1:  PR[GP1:91,2] = PR[GP1:90,2] + 38.566;
   1:L PR[91] R[100]mm/sec CNT100;
   1:  PR[GP1:91,1] = PR[GP1:90,1] + -30.433;
   1:  PR[GP1:91,2] = PR[GP1:90,2] + 38.332;
   1:L PR[91] R[100]mm/sec CNT100;
   1:  PR[GP1:91,1] = PR[GP1:90,1] + -42.580;
   1:  PR[GP1:91,2] = PR[GP1:90,2] + 28.627;
   1:L PR[91] R[100]mm/sec CNT100;
   1:  PR[GP1:91,1] = PR[GP1:90,1] + -42.751;
   1:  PR[GP1:91,2] = PR[GP1:90,2] + 28.506;
   1:L PR[91] R[100]mm/sec CNT100;
   1:  PR[GP1:91,1] = PR[GP1:90,1] + -42.865;
   1:  PR[GP1:91,2] = PR[GP1:90,2] + 28.368;
   1:L PR[91] R[100]mm/sec CNT100;
   1:  PR[GP1:91,1] = PR[GP1:90,1] + -49.282;
   1:  PR[GP1:91,2] = PR[GP1:90,2] + 17.648;
   1:L PR[91] R[100]mm/sec CNT100;
   1:  PR[GP1:91,1] = PR[GP1:90,1] + -50.824;
   1:  PR[GP1:91,2] = PR[GP1:90,2] + 15.096;
   1:L PR[91] R[100]mm/sec CNT100;
   1:  PR[GP1:91,1] = PR[GP1:90,1] + -53.616;
   1:  PR[GP1:91,2] = PR[GP1:90,2] + -0.082;
   1:L PR[91] R[100]mm/sec CNT100;
   1:  PR[GP1:91,1] = PR[GP1:90,1] + -53.593;
   1:  PR[GP1:91,2] = PR[GP1:90,2] + -0.238;
   1:L PR[91] R[100]mm/sec CNT100;
   1:  PR[GP1:91,1] = PR[GP1:90,1] + -50.825;
   1:  PR[GP1:91,2] = PR[GP1:90,2] + -15.238;
   1:L PR[91] R[100]mm/sec CNT100;
   1:  PR[GP1:91,1] = PR[GP1:90,1] + -49.282;
   1:  PR[GP1:91,2] = PR[GP1:90,2] + -17.791;
   1:L PR[91] R[100]mm/sec CNT100;
   1:  PR[GP1:91,1] = PR[GP1:90,1] + -42.867;
   1:  PR[GP1:91,2] = PR[GP1:90,2] + -28.510;
   1:L PR[91] R[100]mm/sec CNT100;
   1:  PR[GP1:91,1] = PR[GP1:90,1] + -42.740;
   1:  PR[GP1:91,2] = PR[GP1:90,2] + -28.662;
   1:L PR[91] R[100]mm/sec CNT100;
   1:  PR[GP1:91,1] = PR[GP1:90,1] + -30.993;
   1:  PR[GP1:91,2] = PR[GP1:90,2] + -38.085;
   1:L PR[91] R[100]mm/sec CNT100;
   1:  PR[GP1:91,1] = PR[GP1:90,1] + -30.452;
   1:  PR[GP1:91,2] = PR[GP1:90,2] + -38.468;
   1:L PR[91] R[100]mm/sec CNT100;
   1:  PR[GP1:91,1] = PR[GP1:90,1] + -29.831;
   1:  PR[GP1:91,2] = PR[GP1:90,2] + -38.709;
   1:L PR[91] R[100]mm/sec CNT100;
   1:  PR[GP1:91,1] = PR[GP1:90,1] + -15.811;
   1:  PR[GP1:91,2] = PR[GP1:90,2] + -43.428;
   1:L PR[91] R[100]mm/sec CNT100;
   1:  PR[GP1:91,1] = PR[GP1:90,1] + -14.631;
   1:  PR[GP1:91,2] = PR[GP1:90,2] + -43.574;
   1:L PR[91] R[100]mm/sec CNT100;
   1:  PR[GP1:91,1] = PR[GP1:90,1] + -0.739;
   1:  PR[GP1:91,2] = PR[GP1:90,2] + -43.223;
   1:L PR[91] R[100]mm/sec CNT100;
   1:  PR[GP1:91,1] = PR[GP1:90,1] + 0.954;
   1:L PR[91] R[100]mm/sec CNT100;
   1:  PR[GP1:91,1] = PR[GP1:90,1] + 14.847;
   1:  PR[GP1:91,2] = PR[GP1:90,2] + -43.574;
   1:L PR[91] R[100]mm/sec CNT100;
   1:  PR[GP1:91,1] = PR[GP1:90,1] + 16.027;
   1:  PR[GP1:91,2] = PR[GP1:90,2] + -43.428;
   1:L PR[91] R[100]mm/sec CNT100;
   1:  PR[GP1:91,1] = PR[GP1:90,1] + 30.046;
   1:  PR[GP1:91,2] = PR[GP1:90,2] + -38.708;
   1:L PR[91] R[100]mm/sec CNT100;
   1:  PR[GP1:91,1] = PR[GP1:90,1] + 30.651;
   1:  PR[GP1:91,2] = PR[GP1:90,2] + -38.474;
   1:L PR[91] R[100]mm/sec CNT100;
   1:  PR[GP1:91,1] = PR[GP1:90,1] + 42.795;
   1:  PR[GP1:91,2] = PR[GP1:90,2] + -28.766;
   1:L PR[91] R[100]mm/sec CNT100;
   1:  PR[GP1:91,1] = PR[GP1:90,1] + 42.966;
   1:  PR[GP1:91,2] = PR[GP1:90,2] + -28.645;
   1:L PR[91] R[100]mm/sec CNT100;
   1:  PR[GP1:91,1] = PR[GP1:90,1] + 43.081;
   1:  PR[GP1:91,2] = PR[GP1:90,2] + -28.507;
   1:L PR[91] R[100]mm/sec CNT100;
   1:  PR[GP1:91,1] = PR[GP1:90,1] + 49.493;
   1:  PR[GP1:91,2] = PR[GP1:90,2] + -17.799;
   1:L PR[91] R[100]mm/sec CNT100;
   1:  PR[GP1:91,1] = PR[GP1:90,1] + 51.038;
   1:  PR[GP1:91,2] = PR[GP1:90,2] + -15.243;
   1:L PR[91] R[100]mm/sec CNT100;
   1:  PR[GP1:91,1] = PR[GP1:90,1] + 53.827;
   1:  PR[GP1:91,2] = PR[GP1:90,2] + -0.072;
   1:L PR[91] R[100]mm/sec CNT100;
   1:  PR[GP1:91,1] = PR[GP1:90,1] + 51.038;
   1:  PR[GP1:91,2] = PR[GP1:90,2] + 15.100;
   1:L PR[91] R[100]mm/sec CNT100;
   1:  PR[GP1:91,1] = PR[GP1:90,1] + 49.493;
   1:  PR[GP1:91,2] = PR[GP1:90,2] + 17.656;
   1:L PR[91] R[100]mm/sec CNT100;
   1:  PR[GP1:91,1] = PR[GP1:90,1] + 43.079;
   1:  PR[GP1:91,2] = PR[GP1:90,2] + 28.365;
   1:L PR[91] R[100]mm/sec CNT100;
   1:  PR[GP1:91,1] = PR[GP1:90,1] + 42.953;
   1:  PR[GP1:91,2] = PR[GP1:90,2] + 28.517;
   1:L PR[91] R[100]mm/sec CNT100;
   1:  PR[GP1:91,1] = PR[GP1:90,1] + 31.205;
   1:  PR[GP1:91,2] = PR[GP1:90,2] + 37.942;
   1:L PR[91] R[100]mm/sec CNT100;
   1:  PR[GP1:91,1] = PR[GP1:90,1] + 30.665;
   1:  PR[GP1:91,2] = PR[GP1:90,2] + 38.325;
   1:L PR[91] R[100]mm/sec CNT100;
   1:  PR[GP1:91,1] = PR[GP1:90,1] + 30.043;
   1:  PR[GP1:91,2] = PR[GP1:90,2] + 38.566;
   1:L PR[91] R[100]mm/sec CNT100;
   1:  PR[GP1:91,1] = PR[GP1:90,1] + 16.023;
   1:  PR[GP1:91,2] = PR[GP1:90,2] + 43.285;
   1:L PR[91] R[100]mm/sec CNT100;
   1:  PR[GP1:91,1] = PR[GP1:90,1] + 14.843;
   1:  PR[GP1:91,2] = PR[GP1:90,2] + 43.431;
   1:L PR[91] R[100]mm/sec CNT100;
   1:  PR[GP1:91,1] = PR[GP1:90,1] + 0.954;
   1:  PR[GP1:91,2] = PR[GP1:90,2] + 43.079;
   1:L PR[91] R[100]mm/sec CNT100;
   1:  ! -- Layer/Ebene 171 -- !;
   1:  PR[91] = PR[90];
   1:  PR[GP1:91,1] = PR[GP1:90,1] + -0.716;
   1:  PR[GP1:91,2] = PR[GP1:90,2] + 43.238;
   1:  PR[GP1:91,3] = PR[GP1:90,3] + 104.615;
   1:L PR[91] R[100]mm/sec CNT100;
   1:  PR[GP1:91,1] = PR[GP1:90,1] + -14.257;
   1:  PR[GP1:91,2] = PR[GP1:90,2] + 43.579;
   1:L PR[91] R[100]mm/sec CNT100;
   1:  PR[GP1:91,1] = PR[GP1:90,1] + -15.711;
   1:  PR[GP1:91,2] = PR[GP1:90,2] + 43.399;
   1:L PR[91] R[100]mm/sec CNT100;
   1:  PR[GP1:91,1] = PR[GP1:90,1] + -29.378;
   1:  PR[GP1:91,2] = PR[GP1:90,2] + 38.799;
   1:L PR[91] R[100]mm/sec CNT100;
   1:  PR[GP1:91,1] = PR[GP1:90,1] + -30.253;
   1:  PR[GP1:91,2] = PR[GP1:90,2] + 38.460;
   1:L PR[91] R[100]mm/sec CNT100;
   1:  PR[GP1:91,1] = PR[GP1:90,1] + -42.093;
   1:  PR[GP1:91,2] = PR[GP1:90,2] + 29.000;
   1:L PR[91] R[100]mm/sec CNT100;
   1:  PR[GP1:91,1] = PR[GP1:90,1] + -42.510;
   1:  PR[GP1:91,2] = PR[GP1:90,2] + 28.705;
   1:L PR[91] R[100]mm/sec CNT100;
   1:  PR[GP1:91,1] = PR[GP1:90,1] + -42.841;
   1:  PR[GP1:91,2] = PR[GP1:90,2] + 28.306;
   1:L PR[91] R[100]mm/sec CNT100;
   1:  PR[GP1:91,1] = PR[GP1:90,1] + -50.650;
   1:  PR[GP1:91,2] = PR[GP1:90,2] + 15.261;
   1:L PR[91] R[100]mm/sec CNT100;
   1:  PR[GP1:91,1] = PR[GP1:90,1] + -50.716;
   1:  PR[GP1:91,2] = PR[GP1:90,2] + 15.111;
   1:L PR[91] R[100]mm/sec CNT100;
   1:  PR[GP1:91,1] = PR[GP1:90,1] + -53.481;
   1:  PR[GP1:91,2] = PR[GP1:90,2] + -0.072;
   1:L PR[91] R[100]mm/sec CNT100;
   1:  PR[GP1:91,1] = PR[GP1:90,1] + -50.739;
   1:  PR[GP1:91,2] = PR[GP1:90,2] + -15.066;
   1:L PR[91] R[100]mm/sec CNT100;
   1:  PR[GP1:91,1] = PR[GP1:90,1] + -50.711;
   1:  PR[GP1:91,2] = PR[GP1:90,2] + -15.266;
   1:L PR[91] R[100]mm/sec CNT100;
   1:  PR[GP1:91,1] = PR[GP1:90,1] + -50.650;
   1:  PR[GP1:91,2] = PR[GP1:90,2] + -15.404;
   1:L PR[91] R[100]mm/sec CNT100;
   1:  PR[GP1:91,1] = PR[GP1:90,1] + -42.843;
   1:  PR[GP1:91,2] = PR[GP1:90,2] + -28.448;
   1:L PR[91] R[100]mm/sec CNT100;
   1:  PR[GP1:91,1] = PR[GP1:90,1] + -42.500;
   1:  PR[GP1:91,2] = PR[GP1:90,2] + -28.861;
   1:L PR[91] R[100]mm/sec CNT100;
   1:  PR[GP1:91,1] = PR[GP1:90,1] + -31.049;
   1:  PR[GP1:91,2] = PR[GP1:90,2] + -38.046;
   1:L PR[91] R[100]mm/sec CNT100;
   1:  PR[GP1:91,1] = PR[GP1:90,1] + -30.272;
   1:  PR[GP1:91,2] = PR[GP1:90,2] + -38.596;
   1:L PR[91] R[100]mm/sec CNT100;
   1:  PR[GP1:91,1] = PR[GP1:90,1] + -29.380;
   1:  PR[GP1:91,2] = PR[GP1:90,2] + -38.942;
   1:L PR[91] R[100]mm/sec CNT100;
   1:  PR[GP1:91,1] = PR[GP1:90,1] + -15.715;
   1:  PR[GP1:91,2] = PR[GP1:90,2] + -43.542;
   1:L PR[91] R[100]mm/sec CNT100;
   1:  PR[GP1:91,1] = PR[GP1:90,1] + -14.261;
   1:  PR[GP1:91,2] = PR[GP1:90,2] + -43.722;
   1:L PR[91] R[100]mm/sec CNT100;
   1:  PR[GP1:91,1] = PR[GP1:90,1] + -0.716;
   1:  PR[GP1:91,2] = PR[GP1:90,2] + -43.382;
   1:L PR[91] R[100]mm/sec CNT100;
   1:  PR[GP1:91,1] = PR[GP1:90,1] + 0.931;
   1:L PR[91] R[100]mm/sec CNT100;
   1:  PR[GP1:91,1] = PR[GP1:90,1] + 14.476;
   1:  PR[GP1:91,2] = PR[GP1:90,2] + -43.722;
   1:L PR[91] R[100]mm/sec CNT100;
   1:  PR[GP1:91,1] = PR[GP1:90,1] + 15.930;
   1:  PR[GP1:91,2] = PR[GP1:90,2] + -43.542;
   1:L PR[91] R[100]mm/sec CNT100;
   1:  PR[GP1:91,1] = PR[GP1:90,1] + 29.595;
   1:  PR[GP1:91,2] = PR[GP1:90,2] + -38.941;
   1:L PR[91] R[100]mm/sec CNT100;
   1:  PR[GP1:91,1] = PR[GP1:90,1] + 30.470;
   1:  PR[GP1:91,2] = PR[GP1:90,2] + -38.602;
   1:L PR[91] R[100]mm/sec CNT100;
   1:  PR[GP1:91,1] = PR[GP1:90,1] + 42.309;
   1:  PR[GP1:91,2] = PR[GP1:90,2] + -29.139;
   1:L PR[91] R[100]mm/sec CNT100;
   1:  PR[GP1:91,1] = PR[GP1:90,1] + 42.726;
   1:  PR[GP1:91,2] = PR[GP1:90,2] + -28.844;
   1:L PR[91] R[100]mm/sec CNT100;
   1:  PR[GP1:91,1] = PR[GP1:90,1] + 43.057;
   1:  PR[GP1:91,2] = PR[GP1:90,2] + -28.445;
   1:L PR[91] R[100]mm/sec CNT100;
   1:  PR[GP1:91,1] = PR[GP1:90,1] + 50.864;
   1:  PR[GP1:91,2] = PR[GP1:90,2] + -15.409;
   1:L PR[91] R[100]mm/sec CNT100;
   1:  PR[GP1:91,1] = PR[GP1:90,1] + 50.930;
   1:  PR[GP1:91,2] = PR[GP1:90,2] + -15.259;
   1:L PR[91] R[100]mm/sec CNT100;
   1:  PR[GP1:91,1] = PR[GP1:90,1] + 53.695;
   1:  PR[GP1:91,2] = PR[GP1:90,2] + -0.072;
   1:L PR[91] R[100]mm/sec CNT100;
   1:  PR[GP1:91,1] = PR[GP1:90,1] + 50.952;
   1:  PR[GP1:91,2] = PR[GP1:90,2] + 14.928;
   1:L PR[91] R[100]mm/sec CNT100;
   1:  PR[GP1:91,1] = PR[GP1:90,1] + 50.924;
   1:  PR[GP1:91,2] = PR[GP1:90,2] + 15.128;
   1:L PR[91] R[100]mm/sec CNT100;
   1:  PR[GP1:91,1] = PR[GP1:90,1] + 50.863;
   1:  PR[GP1:91,2] = PR[GP1:90,2] + 15.266;
   1:L PR[91] R[100]mm/sec CNT100;
   1:  PR[GP1:91,1] = PR[GP1:90,1] + 43.056;
   1:  PR[GP1:91,2] = PR[GP1:90,2] + 28.303;
   1:L PR[91] R[100]mm/sec CNT100;
   1:  PR[GP1:91,1] = PR[GP1:90,1] + 42.713;
   1:  PR[GP1:91,2] = PR[GP1:90,2] + 28.716;
   1:L PR[91] R[100]mm/sec CNT100;
   1:  PR[GP1:91,1] = PR[GP1:90,1] + 31.261;
   1:  PR[GP1:91,2] = PR[GP1:90,2] + 37.903;
   1:L PR[91] R[100]mm/sec CNT100;
   1:  PR[GP1:91,1] = PR[GP1:90,1] + 30.484;
   1:  PR[GP1:91,2] = PR[GP1:90,2] + 38.453;
   1:L PR[91] R[100]mm/sec CNT100;
   1:  PR[GP1:91,1] = PR[GP1:90,1] + 29.593;
   1:  PR[GP1:91,2] = PR[GP1:90,2] + 38.799;
   1:L PR[91] R[100]mm/sec CNT100;
   1:  PR[GP1:91,1] = PR[GP1:90,1] + 15.927;
   1:  PR[GP1:91,2] = PR[GP1:90,2] + 43.399;
   1:L PR[91] R[100]mm/sec CNT100;
   1:  PR[GP1:91,1] = PR[GP1:90,1] + 14.472;
   1:  PR[GP1:91,2] = PR[GP1:90,2] + 43.579;
   1:L PR[91] R[100]mm/sec CNT100;
   1:  PR[GP1:91,1] = PR[GP1:90,1] + 0.931;
   1:  PR[GP1:91,2] = PR[GP1:90,2] + 43.238;
   1:L PR[91] R[100]mm/sec CNT100;
   1:  ! -- Layer/Ebene 172 -- !;
   1:  PR[91] = PR[90];
   1:  PR[GP1:91,1] = PR[GP1:90,1] + -0.694;
   1:  PR[GP1:91,2] = PR[GP1:90,2] + 43.397;
   1:  PR[GP1:91,3] = PR[GP1:90,3] + 105.225;
   1:L PR[91] R[100]mm/sec CNT100;
   1:  PR[GP1:91,1] = PR[GP1:90,1] + -10.734;
   1:  PR[GP1:91,2] = PR[GP1:90,2] + 43.659;
   1:L PR[91] R[100]mm/sec CNT100;
   1:  PR[GP1:91,1] = PR[GP1:90,1] + -13.885;
   1:  PR[GP1:91,2] = PR[GP1:90,2] + 43.727;
   1:L PR[91] R[100]mm/sec CNT100;
   1:  PR[GP1:91,1] = PR[GP1:90,1] + -15.615;
   1:  PR[GP1:91,2] = PR[GP1:90,2] + 43.513;
   1:L PR[91] R[100]mm/sec CNT100;
   1:  PR[GP1:91,1] = PR[GP1:90,1] + -28.928;
   1:  PR[GP1:91,2] = PR[GP1:90,2] + 39.032;
   1:L PR[91] R[100]mm/sec CNT100;
   1:  PR[GP1:91,1] = PR[GP1:90,1] + -30.073;
   1:  PR[GP1:91,2] = PR[GP1:90,2] + 38.589;
   1:L PR[91] R[100]mm/sec CNT100;
   1:  PR[GP1:91,1] = PR[GP1:90,1] + -41.606;
   1:  PR[GP1:91,2] = PR[GP1:90,2] + 29.373;
   1:L PR[91] R[100]mm/sec CNT100;
   1:  PR[GP1:91,1] = PR[GP1:90,1] + -42.270;
   1:  PR[GP1:91,2] = PR[GP1:90,2] + 28.904;
   1:L PR[91] R[100]mm/sec CNT100;
   1:  PR[GP1:91,1] = PR[GP1:90,1] + -42.818;
   1:  PR[GP1:91,2] = PR[GP1:90,2] + 28.244;
   1:L PR[91] R[100]mm/sec CNT100;
   1:  PR[GP1:91,1] = PR[GP1:90,1] + -50.424;
   1:  PR[GP1:91,2] = PR[GP1:90,2] + 15.537;
   1:L PR[91] R[100]mm/sec CNT100;
   1:  PR[GP1:91,1] = PR[GP1:90,1] + -50.631;
   1:  PR[GP1:91,2] = PR[GP1:90,2] + 15.068;
   1:L PR[91] R[100]mm/sec CNT100;
   1:  PR[GP1:91,1] = PR[GP1:90,1] + -53.333;
   1:  PR[GP1:91,2] = PR[GP1:90,2] + 0.249;
   1:L PR[91] R[100]mm/sec CNT100;
   1:  PR[GP1:91,1] = PR[GP1:90,1] + -53.376;
   1:  PR[GP1:91,2] = PR[GP1:90,2] + -0.059;
   1:L PR[91] R[100]mm/sec CNT100;
   1:  PR[GP1:91,1] = PR[GP1:90,1] + -50.702;
   1:  PR[GP1:91,2] = PR[GP1:90,2] + -14.678;
   1:L PR[91] R[100]mm/sec CNT100;
   1:  PR[GP1:91,1] = PR[GP1:90,1] + -50.626;
   1:  PR[GP1:91,2] = PR[GP1:90,2] + -15.223;
   1:L PR[91] R[100]mm/sec CNT100;
   1:  PR[GP1:91,1] = PR[GP1:90,1] + -50.424;
   1:  PR[GP1:91,2] = PR[GP1:90,2] + -15.680;
   1:L PR[91] R[100]mm/sec CNT100;
   1:  PR[GP1:91,1] = PR[GP1:90,1] + -42.819;
   1:  PR[GP1:91,2] = PR[GP1:90,2] + -28.386;
   1:L PR[91] R[100]mm/sec CNT100;
   1:  PR[GP1:91,1] = PR[GP1:90,1] + -42.259;
   1:  PR[GP1:91,2] = PR[GP1:90,2] + -29.060;
   1:L PR[91] R[100]mm/sec CNT100;
   1:  PR[GP1:91,1] = PR[GP1:90,1] + -31.105;
   1:  PR[GP1:91,2] = PR[GP1:90,2] + -38.008;
   1:L PR[91] R[100]mm/sec CNT100;
   1:  PR[GP1:91,1] = PR[GP1:90,1] + -30.092;
   1:  PR[GP1:91,2] = PR[GP1:90,2] + -38.725;
   1:L PR[91] R[100]mm/sec CNT100;
   1:  PR[GP1:91,1] = PR[GP1:90,1] + -28.930;
   1:  PR[GP1:91,2] = PR[GP1:90,2] + -39.175;
   1:L PR[91] R[100]mm/sec CNT100;
   1:  PR[GP1:91,1] = PR[GP1:90,1] + -15.618;
   1:  PR[GP1:91,2] = PR[GP1:90,2] + -43.656;
   1:L PR[91] R[100]mm/sec CNT100;
   1:  PR[GP1:91,1] = PR[GP1:90,1] + -13.889;
   1:  PR[GP1:91,2] = PR[GP1:90,2] + -43.871;
   1:L PR[91] R[100]mm/sec CNT100;
   1:  PR[GP1:91,1] = PR[GP1:90,1] + -10.727;
   1:  PR[GP1:91,2] = PR[GP1:90,2] + -43.803;
   1:L PR[91] R[100]mm/sec CNT100;
   1:  PR[GP1:91,1] = PR[GP1:90,1] + -0.694;
   1:  PR[GP1:91,2] = PR[GP1:90,2] + -43.541;
   1:L PR[91] R[100]mm/sec CNT100;
   1:  PR[GP1:91,1] = PR[GP1:90,1] + 0.909;
   1:L PR[91] R[100]mm/sec CNT100;
   1:  PR[GP1:91,1] = PR[GP1:90,1] + 10.942;
   1:  PR[GP1:91,2] = PR[GP1:90,2] + -43.802;
   1:L PR[91] R[100]mm/sec CNT100;
   1:  PR[GP1:91,1] = PR[GP1:90,1] + 14.104;
   1:  PR[GP1:91,2] = PR[GP1:90,2] + -43.870;
   1:L PR[91] R[100]mm/sec CNT100;
   1:  PR[GP1:91,1] = PR[GP1:90,1] + 15.833;
   1:  PR[GP1:91,2] = PR[GP1:90,2] + -43.656;
   1:L PR[91] R[100]mm/sec CNT100;
   1:  PR[GP1:91,1] = PR[GP1:90,1] + 29.145;
   1:  PR[GP1:91,2] = PR[GP1:90,2] + -39.174;
   1:L PR[91] R[100]mm/sec CNT100;
   1:  PR[GP1:91,1] = PR[GP1:90,1] + 30.290;
   1:  PR[GP1:91,2] = PR[GP1:90,2] + -38.731;
   1:L PR[91] R[100]mm/sec CNT100;
   1:  PR[GP1:91,1] = PR[GP1:90,1] + 41.822;
   1:  PR[GP1:91,2] = PR[GP1:90,2] + -29.513;
   1:L PR[91] R[100]mm/sec CNT100;
   1:  PR[GP1:91,1] = PR[GP1:90,1] + 42.485;
   1:  PR[GP1:91,2] = PR[GP1:90,2] + -29.043;
   1:L PR[91] R[100]mm/sec CNT100;
   1:  PR[GP1:91,1] = PR[GP1:90,1] + 43.033;
   1:  PR[GP1:91,2] = PR[GP1:90,2] + -28.383;
   1:L PR[91] R[100]mm/sec CNT100;
   1:  PR[GP1:91,1] = PR[GP1:90,1] + 50.638;
   1:  PR[GP1:91,2] = PR[GP1:90,2] + -15.685;
   1:L PR[91] R[100]mm/sec CNT100;
   1:  PR[GP1:91,1] = PR[GP1:90,1] + 50.845;
   1:  PR[GP1:91,2] = PR[GP1:90,2] + -15.216;
   1:L PR[91] R[100]mm/sec CNT100;
   1:  PR[GP1:91,1] = PR[GP1:90,1] + 53.546;
   1:  PR[GP1:91,2] = PR[GP1:90,2] + -0.393;
   1:L PR[91] R[100]mm/sec CNT100;
   1:  PR[GP1:91,1] = PR[GP1:90,1] + 53.589;
   1:  PR[GP1:91,2] = PR[GP1:90,2] + -0.085;
   1:L PR[91] R[100]mm/sec CNT100;
   1:  PR[GP1:91,1] = PR[GP1:90,1] + 50.915;
   1:  PR[GP1:91,2] = PR[GP1:90,2] + 14.540;
   1:L PR[91] R[100]mm/sec CNT100;
   1:  PR[GP1:91,1] = PR[GP1:90,1] + 50.839;
   1:  PR[GP1:91,2] = PR[GP1:90,2] + 15.084;
   1:L PR[91] R[100]mm/sec CNT100;
   1:  PR[GP1:91,1] = PR[GP1:90,1] + 50.637;
   1:  PR[GP1:91,2] = PR[GP1:90,2] + 15.542;
   1:L PR[91] R[100]mm/sec CNT100;
   1:  PR[GP1:91,1] = PR[GP1:90,1] + 43.032;
   1:  PR[GP1:91,2] = PR[GP1:90,2] + 28.241;
   1:L PR[91] R[100]mm/sec CNT100;
   1:  PR[GP1:91,1] = PR[GP1:90,1] + 42.472;
   1:  PR[GP1:91,2] = PR[GP1:90,2] + 28.915;
   1:L PR[91] R[100]mm/sec CNT100;
   1:  PR[GP1:91,1] = PR[GP1:90,1] + 31.317;
   1:  PR[GP1:91,2] = PR[GP1:90,2] + 37.864;
   1:L PR[91] R[100]mm/sec CNT100;
   1:  PR[GP1:91,1] = PR[GP1:90,1] + 30.304;
   1:  PR[GP1:91,2] = PR[GP1:90,2] + 38.582;
   1:L PR[91] R[100]mm/sec CNT100;
   1:  PR[GP1:91,1] = PR[GP1:90,1] + 29.142;
   1:  PR[GP1:91,2] = PR[GP1:90,2] + 39.032;
   1:L PR[91] R[100]mm/sec CNT100;
   1:  PR[GP1:91,1] = PR[GP1:90,1] + 15.830;
   1:  PR[GP1:91,2] = PR[GP1:90,2] + 43.513;
   1:L PR[91] R[100]mm/sec CNT100;
   1:  PR[GP1:91,1] = PR[GP1:90,1] + 14.101;
   1:  PR[GP1:91,2] = PR[GP1:90,2] + 43.727;
   1:L PR[91] R[100]mm/sec CNT100;
   1:  PR[GP1:91,1] = PR[GP1:90,1] + 10.949;
   1:  PR[GP1:91,2] = PR[GP1:90,2] + 43.659;
   1:L PR[91] R[100]mm/sec CNT100;
   1:  PR[GP1:91,1] = PR[GP1:90,1] + 0.909;
   1:  PR[GP1:91,2] = PR[GP1:90,2] + 43.397;
   1:L PR[91] R[100]mm/sec CNT100;
   1:  ! -- Layer/Ebene 173 -- !;
   1:  PR[91] = PR[90];
   1:  PR[GP1:91,1] = PR[GP1:90,1] + -0.671;
   1:  PR[GP1:91,2] = PR[GP1:90,2] + 43.557;
   1:  PR[GP1:91,3] = PR[GP1:90,3] + 105.835;
   1:L PR[91] R[100]mm/sec CNT100;
   1:  PR[GP1:91,1] = PR[GP1:90,1] + -9.885;
   1:  PR[GP1:91,2] = PR[GP1:90,2] + 43.797;
   1:L PR[91] R[100]mm/sec CNT100;
   1:  PR[GP1:91,1] = PR[GP1:90,1] + -13.515;
   1:  PR[GP1:91,2] = PR[GP1:90,2] + 43.875;
   1:L PR[91] R[100]mm/sec CNT100;
   1:  PR[GP1:91,1] = PR[GP1:90,1] + -15.518;
   1:  PR[GP1:91,2] = PR[GP1:90,2] + 43.627;
   1:L PR[91] R[100]mm/sec CNT100;
   1:  PR[GP1:91,1] = PR[GP1:90,1] + -28.477;
   1:  PR[GP1:91,2] = PR[GP1:90,2] + 39.265;
   1:L PR[91] R[100]mm/sec CNT100;
   1:  PR[GP1:91,1] = PR[GP1:90,1] + -29.892;
   1:  PR[GP1:91,2] = PR[GP1:90,2] + 38.717;
   1:L PR[91] R[100]mm/sec CNT100;
   1:  PR[GP1:91,1] = PR[GP1:90,1] + -41.120;
   1:  PR[GP1:91,2] = PR[GP1:90,2] + 29.746;
   1:L PR[91] R[100]mm/sec CNT100;
   1:  PR[GP1:91,1] = PR[GP1:90,1] + -42.029;
   1:  PR[GP1:91,2] = PR[GP1:90,2] + 29.102;
   1:L PR[91] R[100]mm/sec CNT100;
   1:  PR[GP1:91,1] = PR[GP1:90,1] + -42.794;
   1:  PR[GP1:91,2] = PR[GP1:90,2] + 28.182;
   1:L PR[91] R[100]mm/sec CNT100;
   1:  PR[GP1:91,1] = PR[GP1:90,1] + -50.198;
   1:  PR[GP1:91,2] = PR[GP1:90,2] + 15.813;
   1:L PR[91] R[100]mm/sec CNT100;
   1:  PR[GP1:91,1] = PR[GP1:90,1] + -50.546;
   1:  PR[GP1:91,2] = PR[GP1:90,2] + 15.025;
   1:L PR[91] R[100]mm/sec CNT100;
   1:  PR[GP1:91,1] = PR[GP1:90,1] + -53.176;
   1:  PR[GP1:91,2] = PR[GP1:90,2] + 0.599;
   1:L PR[91] R[100]mm/sec CNT100;
   1:  PR[GP1:91,1] = PR[GP1:90,1] + -53.268;
   1:  PR[GP1:91,2] = PR[GP1:90,2] + -0.059;
   1:L PR[91] R[100]mm/sec CNT100;
   1:  PR[GP1:91,1] = PR[GP1:90,1] + -50.665;
   1:  PR[GP1:91,2] = PR[GP1:90,2] + -14.289;
   1:L PR[91] R[100]mm/sec CNT100;
   1:  PR[GP1:91,1] = PR[GP1:90,1] + -50.541;
   1:  PR[GP1:91,2] = PR[GP1:90,2] + -15.179;
   1:L PR[91] R[100]mm/sec CNT100;
   1:  PR[GP1:91,1] = PR[GP1:90,1] + -50.198;
   1:  PR[GP1:91,2] = PR[GP1:90,2] + -15.956;
   1:L PR[91] R[100]mm/sec CNT100;
   1:  PR[GP1:91,1] = PR[GP1:90,1] + -42.795;
   1:  PR[GP1:91,2] = PR[GP1:90,2] + -28.324;
   1:L PR[91] R[100]mm/sec CNT100;
   1:  PR[GP1:91,1] = PR[GP1:90,1] + -42.019;
   1:  PR[GP1:91,2] = PR[GP1:90,2] + -29.259;
   1:L PR[91] R[100]mm/sec CNT100;
   1:  PR[GP1:91,1] = PR[GP1:90,1] + -31.161;
   1:  PR[GP1:91,2] = PR[GP1:90,2] + -37.969;
   1:L PR[91] R[100]mm/sec CNT100;
   1:  PR[GP1:91,1] = PR[GP1:90,1] + -29.911;
   1:  PR[GP1:91,2] = PR[GP1:90,2] + -38.853;
   1:L PR[91] R[100]mm/sec CNT100;
   1:  PR[GP1:91,1] = PR[GP1:90,1] + -28.480;
   1:  PR[GP1:91,2] = PR[GP1:90,2] + -39.408;
   1:L PR[91] R[100]mm/sec CNT100;
   1:  PR[GP1:91,1] = PR[GP1:90,1] + -15.521;
   1:  PR[GP1:91,2] = PR[GP1:90,2] + -43.770;
   1:L PR[91] R[100]mm/sec CNT100;
   1:  PR[GP1:91,1] = PR[GP1:90,1] + -13.518;
   1:  PR[GP1:91,2] = PR[GP1:90,2] + -44.019;
   1:L PR[91] R[100]mm/sec CNT100;
   1:  PR[GP1:91,1] = PR[GP1:90,1] + -9.877;
   1:  PR[GP1:91,2] = PR[GP1:90,2] + -43.940;
   1:L PR[91] R[100]mm/sec CNT100;
   1:  PR[GP1:91,1] = PR[GP1:90,1] + -0.671;
   1:  PR[GP1:91,2] = PR[GP1:90,2] + -43.701;
   1:L PR[91] R[100]mm/sec CNT100;
   1:  PR[GP1:91,1] = PR[GP1:90,1] + 0.886;
   1:L PR[91] R[100]mm/sec CNT100;
   1:  PR[GP1:91,1] = PR[GP1:90,1] + 10.092;
   1:  PR[GP1:91,2] = PR[GP1:90,2] + -43.940;
   1:L PR[91] R[100]mm/sec CNT100;
   1:  PR[GP1:91,1] = PR[GP1:90,1] + 13.733;
   1:  PR[GP1:91,2] = PR[GP1:90,2] + -44.018;
   1:L PR[91] R[100]mm/sec CNT100;
   1:  PR[GP1:91,1] = PR[GP1:90,1] + 15.736;
   1:  PR[GP1:91,2] = PR[GP1:90,2] + -43.770;
   1:L PR[91] R[100]mm/sec CNT100;
   1:  PR[GP1:91,1] = PR[GP1:90,1] + 28.694;
   1:  PR[GP1:91,2] = PR[GP1:90,2] + -39.408;
   1:L PR[91] R[100]mm/sec CNT100;
   1:  PR[GP1:91,1] = PR[GP1:90,1] + 30.109;
   1:  PR[GP1:91,2] = PR[GP1:90,2] + -38.859;
   1:L PR[91] R[100]mm/sec CNT100;
   1:  PR[GP1:91,1] = PR[GP1:90,1] + 41.335;
   1:  PR[GP1:91,2] = PR[GP1:90,2] + -29.886;
   1:L PR[91] R[100]mm/sec CNT100;
   1:  PR[GP1:91,1] = PR[GP1:90,1] + 42.245;
   1:  PR[GP1:91,2] = PR[GP1:90,2] + -29.242;
   1:L PR[91] R[100]mm/sec CNT100;
   1:  PR[GP1:91,1] = PR[GP1:90,1] + 43.009;
   1:  PR[GP1:91,2] = PR[GP1:90,2] + -28.321;
   1:L PR[91] R[100]mm/sec CNT100;
   1:  PR[GP1:91,1] = PR[GP1:90,1] + 50.412;
   1:  PR[GP1:91,2] = PR[GP1:90,2] + -15.960;
   1:L PR[91] R[100]mm/sec CNT100;
   1:  PR[GP1:91,1] = PR[GP1:90,1] + 50.759;
   1:  PR[GP1:91,2] = PR[GP1:90,2] + -15.172;
   1:L PR[91] R[100]mm/sec CNT100;
   1:  PR[GP1:91,1] = PR[GP1:90,1] + 53.389;
   1:  PR[GP1:91,2] = PR[GP1:90,2] + -0.743;
   1:L PR[91] R[100]mm/sec CNT100;
   1:  PR[GP1:91,1] = PR[GP1:90,1] + 53.481;
   1:  PR[GP1:91,2] = PR[GP1:90,2] + -0.085;
   1:L PR[91] R[100]mm/sec CNT100;
   1:  PR[GP1:91,1] = PR[GP1:90,1] + 50.878;
   1:  PR[GP1:91,2] = PR[GP1:90,2] + 14.151;
   1:L PR[91] R[100]mm/sec CNT100;
   1:  PR[GP1:91,1] = PR[GP1:90,1] + 50.754;
   1:  PR[GP1:91,2] = PR[GP1:90,2] + 15.041;
   1:L PR[91] R[100]mm/sec CNT100;
   1:  PR[GP1:91,1] = PR[GP1:90,1] + 50.411;
   1:  PR[GP1:91,2] = PR[GP1:90,2] + 15.817;
   1:L PR[91] R[100]mm/sec CNT100;
   1:  PR[GP1:91,1] = PR[GP1:90,1] + 43.008;
   1:  PR[GP1:91,2] = PR[GP1:90,2] + 28.179;
   1:L PR[91] R[100]mm/sec CNT100;
   1:  PR[GP1:91,1] = PR[GP1:90,1] + 42.232;
   1:  PR[GP1:91,2] = PR[GP1:90,2] + 29.114;
   1:L PR[91] R[100]mm/sec CNT100;
   1:  PR[GP1:91,1] = PR[GP1:90,1] + 31.373;
   1:  PR[GP1:91,2] = PR[GP1:90,2] + 37.826;
   1:L PR[91] R[100]mm/sec CNT100;
   1:  PR[GP1:91,1] = PR[GP1:90,1] + 30.124;
   1:  PR[GP1:91,2] = PR[GP1:90,2] + 38.710;
   1:L PR[91] R[100]mm/sec CNT100;
   1:  PR[GP1:91,1] = PR[GP1:90,1] + 28.692;
   1:  PR[GP1:91,2] = PR[GP1:90,2] + 39.265;
   1:L PR[91] R[100]mm/sec CNT100;
   1:  PR[GP1:91,1] = PR[GP1:90,1] + 15.733;
   1:  PR[GP1:91,2] = PR[GP1:90,2] + 43.627;
   1:L PR[91] R[100]mm/sec CNT100;
   1:  PR[GP1:91,1] = PR[GP1:90,1] + 13.730;
   1:  PR[GP1:91,2] = PR[GP1:90,2] + 43.875;
   1:L PR[91] R[100]mm/sec CNT100;
   1:  PR[GP1:91,1] = PR[GP1:90,1] + 10.101;
   1:  PR[GP1:91,2] = PR[GP1:90,2] + 43.797;
   1:L PR[91] R[100]mm/sec CNT100;
   1:  PR[GP1:91,1] = PR[GP1:90,1] + 0.886;
   1:  PR[GP1:91,2] = PR[GP1:90,2] + 43.557;
   1:L PR[91] R[100]mm/sec CNT100;
   1:  ! -- Layer/Ebene 174 -- !;
   1:  PR[91] = PR[90];
   1:  PR[GP1:91,1] = PR[GP1:90,1] + -0.649;
   1:  PR[GP1:91,2] = PR[GP1:90,2] + 43.716;
   1:  PR[GP1:91,3] = PR[GP1:90,3] + 106.445;
   1:L PR[91] R[100]mm/sec CNT100;
   1:  PR[GP1:91,1] = PR[GP1:90,1] + -9.037;
   1:  PR[GP1:91,2] = PR[GP1:90,2] + 43.935;
   1:L PR[91] R[100]mm/sec CNT100;
   1:  PR[GP1:91,1] = PR[GP1:90,1] + -13.144;
   1:  PR[GP1:91,2] = PR[GP1:90,2] + 44.023;
   1:L PR[91] R[100]mm/sec CNT100;
   1:  PR[GP1:91,1] = PR[GP1:90,1] + -15.421;
   1:  PR[GP1:91,2] = PR[GP1:90,2] + 43.741;
   1:L PR[91] R[100]mm/sec CNT100;
   1:  PR[GP1:91,1] = PR[GP1:90,1] + -28.027;
   1:  PR[GP1:91,2] = PR[GP1:90,2] + 39.499;
   1:L PR[91] R[100]mm/sec CNT100;
   1:  PR[GP1:91,1] = PR[GP1:90,1] + -29.712;
   1:  PR[GP1:91,2] = PR[GP1:90,2] + 38.846;
   1:L PR[91] R[100]mm/sec CNT100;
   1:  PR[GP1:91,1] = PR[GP1:90,1] + -40.633;
   1:  PR[GP1:91,2] = PR[GP1:90,2] + 30.120;
   1:L PR[91] R[100]mm/sec CNT100;
   1:  PR[GP1:91,1] = PR[GP1:90,1] + -41.789;
   1:  PR[GP1:91,2] = PR[GP1:90,2] + 29.301;
   1:L PR[91] R[100]mm/sec CNT100;
   1:  PR[GP1:91,1] = PR[GP1:90,1] + -42.770;
   1:  PR[GP1:91,2] = PR[GP1:90,2] + 28.120;
   1:L PR[91] R[100]mm/sec CNT100;
   1:  PR[GP1:91,1] = PR[GP1:90,1] + -49.972;
   1:  PR[GP1:91,2] = PR[GP1:90,2] + 16.089;
   1:L PR[91] R[100]mm/sec CNT100;
   1:  PR[GP1:91,1] = PR[GP1:90,1] + -50.460;
   1:  PR[GP1:91,2] = PR[GP1:90,2] + 14.981;
   1:L PR[91] R[100]mm/sec CNT100;
   1:  PR[GP1:91,1] = PR[GP1:90,1] + -53.019;
   1:  PR[GP1:91,2] = PR[GP1:90,2] + 0.950;
   1:L PR[91] R[100]mm/sec CNT100;
   1:  PR[GP1:91,1] = PR[GP1:90,1] + -53.159;
   1:  PR[GP1:91,2] = PR[GP1:90,2] + -0.059;
   1:L PR[91] R[100]mm/sec CNT100;
   1:  PR[GP1:91,1] = PR[GP1:90,1] + -50.628;
   1:  PR[GP1:91,2] = PR[GP1:90,2] + -13.901;
   1:L PR[91] R[100]mm/sec CNT100;
   1:  PR[GP1:91,1] = PR[GP1:90,1] + -50.456;
   1:  PR[GP1:91,2] = PR[GP1:90,2] + -15.136;
   1:L PR[91] R[100]mm/sec CNT100;
   1:  PR[GP1:91,1] = PR[GP1:90,1] + -49.972;
   1:  PR[GP1:91,2] = PR[GP1:90,2] + -16.232;
   1:L PR[91] R[100]mm/sec CNT100;
   1:  PR[GP1:91,1] = PR[GP1:90,1] + -42.771;
   1:  PR[GP1:91,2] = PR[GP1:90,2] + -28.262;
   1:L PR[91] R[100]mm/sec CNT100;
   1:  PR[GP1:91,1] = PR[GP1:90,1] + -41.778;
   1:  PR[GP1:91,2] = PR[GP1:90,2] + -29.458;
   1:L PR[91] R[100]mm/sec CNT100;
   1:  PR[GP1:91,1] = PR[GP1:90,1] + -31.217;
   1:  PR[GP1:91,2] = PR[GP1:90,2] + -37.930;
   1:L PR[91] R[100]mm/sec CNT100;
   1:  PR[GP1:91,1] = PR[GP1:90,1] + -29.731;
   1:  PR[GP1:91,2] = PR[GP1:90,2] + -38.982;
   1:L PR[91] R[100]mm/sec CNT100;
   1:  PR[GP1:91,1] = PR[GP1:90,1] + -28.029;
   1:  PR[GP1:91,2] = PR[GP1:90,2] + -39.641;
   1:L PR[91] R[100]mm/sec CNT100;
   1:  PR[GP1:91,1] = PR[GP1:90,1] + -15.425;
   1:  PR[GP1:91,2] = PR[GP1:90,2] + -43.884;
   1:L PR[91] R[100]mm/sec CNT100;
   1:  PR[GP1:91,1] = PR[GP1:90,1] + -13.148;
   1:  PR[GP1:91,2] = PR[GP1:90,2] + -44.167;
   1:L PR[91] R[100]mm/sec CNT100;
   1:  PR[GP1:91,1] = PR[GP1:90,1] + -9.027;
   1:  PR[GP1:91,2] = PR[GP1:90,2] + -44.078;
   1:L PR[91] R[100]mm/sec CNT100;
   1:  PR[GP1:91,1] = PR[GP1:90,1] + -0.649;
   1:  PR[GP1:91,2] = PR[GP1:90,2] + -43.860;
   1:L PR[91] R[100]mm/sec CNT100;
   1:  PR[GP1:91,1] = PR[GP1:90,1] + 0.863;
   1:L PR[91] R[100]mm/sec CNT100;
   1:  PR[GP1:91,1] = PR[GP1:90,1] + 9.241;
   1:  PR[GP1:91,2] = PR[GP1:90,2] + -44.078;
   1:L PR[91] R[100]mm/sec CNT100;
   1:  PR[GP1:91,1] = PR[GP1:90,1] + 13.362;
   1:  PR[GP1:91,2] = PR[GP1:90,2] + -44.166;
   1:L PR[91] R[100]mm/sec CNT100;
   1:  PR[GP1:91,1] = PR[GP1:90,1] + 15.640;
   1:  PR[GP1:91,2] = PR[GP1:90,2] + -43.884;
   1:L PR[91] R[100]mm/sec CNT100;
   1:  PR[GP1:91,1] = PR[GP1:90,1] + 28.244;
   1:  PR[GP1:91,2] = PR[GP1:90,2] + -39.641;
   1:L PR[91] R[100]mm/sec CNT100;
   1:  PR[GP1:91,1] = PR[GP1:90,1] + 29.929;
   1:  PR[GP1:91,2] = PR[GP1:90,2] + -38.988;
   1:L PR[91] R[100]mm/sec CNT100;
   1:  PR[GP1:91,1] = PR[GP1:90,1] + 40.848;
   1:  PR[GP1:91,2] = PR[GP1:90,2] + -30.260;
   1:L PR[91] R[100]mm/sec CNT100;
   1:  PR[GP1:91,1] = PR[GP1:90,1] + 42.004;
   1:  PR[GP1:91,2] = PR[GP1:90,2] + -29.441;
   1:L PR[91] R[100]mm/sec CNT100;
   1:  PR[GP1:91,1] = PR[GP1:90,1] + 42.985;
   1:  PR[GP1:91,2] = PR[GP1:90,2] + -28.260;
   1:L PR[91] R[100]mm/sec CNT100;
   1:  PR[GP1:91,1] = PR[GP1:90,1] + 50.185;
   1:  PR[GP1:91,2] = PR[GP1:90,2] + -16.236;
   1:L PR[91] R[100]mm/sec CNT100;
   1:  PR[GP1:91,1] = PR[GP1:90,1] + 50.674;
   1:  PR[GP1:91,2] = PR[GP1:90,2] + -15.129;
   1:L PR[91] R[100]mm/sec CNT100;
   1:  PR[GP1:91,1] = PR[GP1:90,1] + 53.232;
   1:  PR[GP1:91,2] = PR[GP1:90,2] + -1.094;
   1:L PR[91] R[100]mm/sec CNT100;
   1:  PR[GP1:91,1] = PR[GP1:90,1] + 53.373;
   1:  PR[GP1:91,2] = PR[GP1:90,2] + -0.085;
   1:L PR[91] R[100]mm/sec CNT100;
   1:  PR[GP1:91,1] = PR[GP1:90,1] + 50.841;
   1:  PR[GP1:91,2] = PR[GP1:90,2] + 13.762;
   1:L PR[91] R[100]mm/sec CNT100;
   1:  PR[GP1:91,1] = PR[GP1:90,1] + 50.669;
   1:  PR[GP1:91,2] = PR[GP1:90,2] + 14.997;
   1:L PR[91] R[100]mm/sec CNT100;
   1:  PR[GP1:91,1] = PR[GP1:90,1] + 50.185;
   1:  PR[GP1:91,2] = PR[GP1:90,2] + 16.093;
   1:L PR[91] R[100]mm/sec CNT100;
   1:  PR[GP1:91,1] = PR[GP1:90,1] + 42.984;
   1:  PR[GP1:91,2] = PR[GP1:90,2] + 28.117;
   1:L PR[91] R[100]mm/sec CNT100;
   1:  PR[GP1:91,1] = PR[GP1:90,1] + 41.992;
   1:  PR[GP1:91,2] = PR[GP1:90,2] + 29.312;
   1:L PR[91] R[100]mm/sec CNT100;
   1:  PR[GP1:91,1] = PR[GP1:90,1] + 31.429;
   1:  PR[GP1:91,2] = PR[GP1:90,2] + 37.787;
   1:L PR[91] R[100]mm/sec CNT100;
   1:  PR[GP1:91,1] = PR[GP1:90,1] + 29.943;
   1:  PR[GP1:91,2] = PR[GP1:90,2] + 38.839;
   1:L PR[91] R[100]mm/sec CNT100;
   1:  PR[GP1:91,1] = PR[GP1:90,1] + 28.242;
   1:  PR[GP1:91,2] = PR[GP1:90,2] + 39.498;
   1:L PR[91] R[100]mm/sec CNT100;
   1:  PR[GP1:91,1] = PR[GP1:90,1] + 15.636;
   1:  PR[GP1:91,2] = PR[GP1:90,2] + 43.741;
   1:L PR[91] R[100]mm/sec CNT100;
   1:  PR[GP1:91,1] = PR[GP1:90,1] + 13.359;
   1:  PR[GP1:91,2] = PR[GP1:90,2] + 44.023;
   1:L PR[91] R[100]mm/sec CNT100;
   1:  PR[GP1:91,1] = PR[GP1:90,1] + 9.252;
   1:  PR[GP1:91,2] = PR[GP1:90,2] + 43.935;
   1:L PR[91] R[100]mm/sec CNT100;
   1:  PR[GP1:91,1] = PR[GP1:90,1] + 0.863;
   1:  PR[GP1:91,2] = PR[GP1:90,2] + 43.716;
   1:L PR[91] R[100]mm/sec CNT100;
   1:  ! -- Layer/Ebene 175 -- !;
   1:  PR[91] = PR[90];
   1:  PR[GP1:91,1] = PR[GP1:90,1] + -0.626;
   1:  PR[GP1:91,2] = PR[GP1:90,2] + 43.875;
   1:  PR[GP1:91,3] = PR[GP1:90,3] + 107.055;
   1:L PR[91] R[100]mm/sec CNT100;
   1:  PR[GP1:91,1] = PR[GP1:90,1] + -8.188;
   1:  PR[GP1:91,2] = PR[GP1:90,2] + 44.072;
   1:L PR[91] R[100]mm/sec CNT100;
   1:  PR[GP1:91,1] = PR[GP1:90,1] + -12.774;
   1:  PR[GP1:91,2] = PR[GP1:90,2] + 44.171;
   1:L PR[91] R[100]mm/sec CNT100;
   1:  PR[GP1:91,1] = PR[GP1:90,1] + -15.325;
   1:  PR[GP1:91,2] = PR[GP1:90,2] + 43.855;
   1:L PR[91] R[100]mm/sec CNT100;
   1:  PR[GP1:91,1] = PR[GP1:90,1] + -27.577;
   1:  PR[GP1:91,2] = PR[GP1:90,2] + 39.732;
   1:L PR[91] R[100]mm/sec CNT100;
   1:  PR[GP1:91,1] = PR[GP1:90,1] + -29.532;
   1:  PR[GP1:91,2] = PR[GP1:90,2] + 38.974;
   1:L PR[91] R[100]mm/sec CNT100;
   1:  PR[GP1:91,1] = PR[GP1:90,1] + -40.146;
   1:  PR[GP1:91,2] = PR[GP1:90,2] + 30.493;
   1:L PR[91] R[100]mm/sec CNT100;
   1:  PR[GP1:91,1] = PR[GP1:90,1] + -41.548;
   1:  PR[GP1:91,2] = PR[GP1:90,2] + 29.500;
   1:L PR[91] R[100]mm/sec CNT100;
   1:  PR[GP1:91,1] = PR[GP1:90,1] + -42.746;
   1:  PR[GP1:91,2] = PR[GP1:90,2] + 28.058;
   1:L PR[91] R[100]mm/sec CNT100;
   1:  PR[GP1:91,1] = PR[GP1:90,1] + -49.746;
   1:  PR[GP1:91,2] = PR[GP1:90,2] + 16.364;
   1:L PR[91] R[100]mm/sec CNT100;
   1:  PR[GP1:91,1] = PR[GP1:90,1] + -50.375;
   1:  PR[GP1:91,2] = PR[GP1:90,2] + 14.938;
   1:L PR[91] R[100]mm/sec CNT100;
   1:  PR[GP1:91,1] = PR[GP1:90,1] + -52.862;
   1:  PR[GP1:91,2] = PR[GP1:90,2] + 1.301;
   1:L PR[91] R[100]mm/sec CNT100;
   1:  PR[GP1:91,1] = PR[GP1:90,1] + -53.051;
   1:  PR[GP1:91,2] = PR[GP1:90,2] + -0.059;
   1:L PR[91] R[100]mm/sec CNT100;
   1:  PR[GP1:91,1] = PR[GP1:90,1] + -50.591;
   1:  PR[GP1:91,2] = PR[GP1:90,2] + -13.512;
   1:L PR[91] R[100]mm/sec CNT100;
   1:  PR[GP1:91,1] = PR[GP1:90,1] + -50.370;
   1:  PR[GP1:91,2] = PR[GP1:90,2] + -15.093;
   1:L PR[91] R[100]mm/sec CNT100;
   1:  PR[GP1:91,1] = PR[GP1:90,1] + -49.746;
   1:  PR[GP1:91,2] = PR[GP1:90,2] + -16.507;
   1:L PR[91] R[100]mm/sec CNT100;
   1:  PR[GP1:91,1] = PR[GP1:90,1] + -42.747;
   1:  PR[GP1:91,2] = PR[GP1:90,2] + -28.200;
   1:L PR[91] R[100]mm/sec CNT100;
   1:  PR[GP1:91,1] = PR[GP1:90,1] + -41.538;
   1:  PR[GP1:91,2] = PR[GP1:90,2] + -29.657;
   1:L PR[91] R[100]mm/sec CNT100;
   1:  PR[GP1:91,1] = PR[GP1:90,1] + -31.272;
   1:  PR[GP1:91,2] = PR[GP1:90,2] + -37.891;
   1:L PR[91] R[100]mm/sec CNT100;
   1:  PR[GP1:91,1] = PR[GP1:90,1] + -29.551;
   1:  PR[GP1:91,2] = PR[GP1:90,2] + -39.110;
   1:L PR[91] R[100]mm/sec CNT100;
   1:  PR[GP1:91,1] = PR[GP1:90,1] + -27.579;
   1:  PR[GP1:91,2] = PR[GP1:90,2] + -39.874;
   1:L PR[91] R[100]mm/sec CNT100;
   1:  PR[GP1:91,1] = PR[GP1:90,1] + -15.328;
   1:  PR[GP1:91,2] = PR[GP1:90,2] + -43.999;
   1:L PR[91] R[100]mm/sec CNT100;
   1:  PR[GP1:91,1] = PR[GP1:90,1] + -12.777;
   1:  PR[GP1:91,2] = PR[GP1:90,2] + -44.315;
   1:L PR[91] R[100]mm/sec CNT100;
   1:  PR[GP1:91,1] = PR[GP1:90,1] + -8.176;
   1:  PR[GP1:91,2] = PR[GP1:90,2] + -44.216;
   1:L PR[91] R[100]mm/sec CNT100;
